(* CoDeSys 2.3.9.42 project: PLC.pro *)
(* Libraries: STANDARD.LIB 5.6.98 12:03:02, TcBase.lib 14.5.09 12:14:08, TcSystem.lib 21.1.15 10:22:54, TcBaseMath.lib 27.7.04 12:07:56, TcMath.lib 23.9.04 15:15:30, TcMC2.lib 6.5.15 08:29:24, TcUtilities.lib 6.1.15 16:45:04, SysLibAlarmTrend.lib 17.10.05 13:12:38 *)

(* Task configuration *)
TASK Standard (PRIORITY := 0, INTERVAL := T#10ms);
	MAIN
END_TASK

(* Global variable list: Global_Variables *)
VAR_GLOBAL
	Flag_FPC_Brd_Err:BOOL;
	Flag_Robot_Alarm:BOOL;

	Total_PauseStatus:BOOL;(*暂停状态*)

	AA: FB_BasicPID;
	MM: BOOL;
	a1: LREAL;
	a2: LREAL;
	OUTPUT:LREAL;

	Process_2_Can_Push2: BOOL;
	Process_2_Can_Push1: BOOL;


	Save_Par:FB_WritePersistentData;
	Save_Button:BOOL;

	Liftin_Feed_1_Run:BOOL;(*喂料1运行触发*)
	Liftin_Feed_Left_1_Run:BOOL;(*喂料1运行触发*)
	Liftin_Feed_Left_2_Run:BOOL;(*喂料1运行触发*)
	Liftin_Feed_Right_1_Run:BOOL;(*喂料1运行触发*)
	Liftin_Feed_Right_2_Run:BOOL;(*喂料1运行触发*)
	Left_Carry_Run:BOOL;(*左搬运*)
	PC_Pause:BOOL;(*上位机给我暂停*)

	Right_Carry_Run:BOOL;(*左搬运*)
	Product_Film_Handel_Run:BOOL;(*吸膜撕膜位置工作触发*)

	Left_Translation_Run:BOOL;(*左平移运行触发*)
	Left_Translation_Run_1: BOOL;
	Left_Translation_Run_2: BOOL;

	Right_Translation_Run:BOOL;(*右平移运动触发*)
	Rolling_Part_Run:BOOL;(*滚压运行触发*)


(*初始化进程*)
	IniRun_Run:BOOL;(*初始化进程触发*)(*-----------------未用-----------------------------*)
	Model_Choose:BOOL;(*模式选择状态*)
	Need_Ini:BOOL;(*需要初始化*)
	IsIniing:BOOL;(*	初始化中*)
	home_backing:BOOL;(*回原点中*)
	runing: BOOL;(*运行中*)

(*上料升降状态信息*)
	Feed_1_Finish:BOOL;(*上料喂料1完成------to上料流程*)

(*撕膜流程为流程1---------------------左移载为流程2--------------------------*)

(*撕膜流程位置状态标志位*)

	Tray1_Have: BOOL; (*1料盘有料*)
	Tray2_Have: BOOL;(*2料盘有料*)

	Process_1_Get_Finish:BOOL;(*喂料1-----拿到料完成----to feed1*)


	Process_1_Push_Finish:BOOL;(*放料完成-----to流程2*)
	Process_1_Push_Finish_Sure:BOOL;(*放料完成-----to流程2*)


	Process_2_Can_Push:BOOL;(*TO---流程1*)

	Positive1_Safe:BOOL;
	Positive2_Safe:BOOL;
	Positive3_Safe:BOOL;
	Positive4_Safe:BOOL;
	Positive_Wait_Safe:BOOL;
(*1------------------------------------------------2*)
(*1------------------------------------------------1*)
(*1------------------------------------------------1*)
(*1------------------------------------------------1*)
(*1------------------------------------------------1*)
(*1------------------------------------------------1*)
(*1------------------------------------------------1*)
(*4------------------------------------------------3*)

	Positive_Camera_Safe1:BOOL;(*拍照位置1安全*)
	Positive_Camera_Safe2:BOOL;(*拍照位置1安全*)
	Positive_Camera_Safe3:BOOL;(*拍照位置1安全*)
	Positive_Camera_Safe4: BOOL;	(* (*拍照位置1安全*) *)

	Positive_Fit_Safe1:BOOL;(*贴合位置1安全*)
	Positive_Fit_Safe2:BOOL;(*贴合位置1安全*)
	Positive_Fit_Safe3:BOOL;(*贴合位置1安全*)
	Positive_Fit_Safe4:BOOL;(*贴合位置1安全*)







	Process_2_Set_Finish1: BOOL;
	Process_2_Set_Finish2: BOOL;

	Wait_Robort2_Touch_Finish:BOOL;(*机械手2贴合完成，关真空吸*)

	Get_Robot1_Get_Finish:BOOL;(*机械手1对取料贴合完成，左移载可动作-------From   机械手1*)
	Robot2_Push_Finish:BOOL;(*机械手2----放料到滚压完成*)

	Feed_2_Finish:BOOL;(*111111111上料喂料2完成 ------TO 机械手1*)
	Get_Robot1_Tray_Empty:BOOL;(*2222222222机械手1取料盘空信号  -------From  机械手1*)
	zuo_ke_jiang:BOOL;(*5555555左可下降*)
	zuo_down_Finish:BOOL;(*1111111判断是否可放*)
	Left_Can_Move: BOOL;(*3333333可以移动*)
	Left_Move_Finish:BOOL;(*4444444移动完成*)

	Feed_3_Finish:BOOL;(*上料喂料3完成------to   机械手3*)
	Get_Robort3_Tray_Full:BOOL;(*机械手3给出，右升降料盘空*)

	Right_Loading_OK:BOOL;(*上空盘ok*)
	Right_Get_Tray_OK:BOOL;(*取空盘完成*)
	Right_Need_Tray:BOOL;(*要空盘信号*)
	Right_Send_Tray_OK:BOOL;(*上空盘完成*)

	you_down_Finish: BOOL;
	you_ke_jiang: BOOL;
	Right_Can_Move:BOOL;
	Right_Move_Finish:BOOL;



(*滚压流程3---------------------------------------右移载流程4*)

	Process_3_Can_Push:BOOL;(*滚压可放料------to 机械收2*)
	Wait_Robot_Push:BOOL;(*机械手放滚压，开真空吸*)
  	Process_3_Set_Finish:BOOL;(*滚压送出料----完成信号*)

	Process_4_Can_Push:BOOL;(*右移载可放料-------to 滚压流程*)
	Process_4_Set_Finish:BOOL;(*右移载，到位，机械手3可操作------to 机械手3*)
	Get_Robort_simo_Finish: BOOL;(*获取机械手撕膜完成信号*)
	Set_Robort_Can_Get: BOOL;(*告知机械手可取料*)


	Get_Robot3_Get_Finish:BOOL;(*机械手3----给出，取右移载完成信号*)



(*界面按钮*)
	Silencer_Button: BOOL;(*消音按钮*)
	Discharge_Button:BOOL;(*排料按钮*)

	UP_Button:BOOL;(*上料按钮*)
	Left_UP_Button:BOOL;(*左上料按钮*)
	Left_Down_Button:BOOL;(*右卸料按钮*)

	Right_UP_Button:BOOL;(*右上料按钮*)
	Right_Down_Button:BOOL;(*右卸料按钮*)

	Button_Ad:BOOL;

	Feed1_Button:BOOL;(*上料自动按钮*)
	Feed_Left_Button1:BOOL;(*左上升自动按钮*)
	Feed_Left_Button2:BOOL;(*左下降自动按钮*)
	Feed_Right_Button1:BOOL;(*右上升自动按钮*)
	Feed_Right_Button2:BOOL;(*右下降自动按钮*)





(*显示运行状态*)




(*显示报警*)


(*标志位1*)
	shou_have_mo:BOOL;(*有膜*)
	shou_have_moliao:BOOL;(*有膜料*)
	shou_have_liao:BOOL;(*有料*)
	zai_have_liao:BOOL;(*载盘有料*)
	zai_have_mo:BOOL;(*载盘有膜*)


(*接收机械手完成信号*)
	Camera_1_1_OK:BOOL;(*已拍照1-----FROM JIXIESHOU*)
	Camera_1_2_OK:BOOL;(*已拍照2-----FROM JIXIESHOU*)
	Camera_1_3_OK:BOOL;(*已拍照3-----FROM JIXIESHOU*)
	Camera_1_4_OK:BOOL;(*已拍照4-----FROM JIXIESHOU*)

	Camera_2_1_OK:BOOL;(*已拍照1-----FROM JIXIESHOU*)
	Camera_2_2_OK:BOOL;(*已拍照2-----FROM JIXIESHOU*)



(*左流程，运行触发----发送给机械手*)
	Camera_1_1_run:BOOL;(*拍照1标志位-----TO JIXIESOU*)
	Camera_1_2_run:BOOL;(*拍照2标志位----TO JIXIESOU*)
	Camera_1_3_run:BOOL;(*拍照3标志位----TO JIXIESOU*)
	Camera_1_4_run:BOOL;(*拍照4标志位----TO JIXIESOU*)
	Camera_2_1_run:BOOL;(*拍照1标志位-----TO JIXIESOU*)
	Camera_2_2_run:BOOL;(*拍照2标志位----TO JIXIESOU*)

	Camera_1_5_run: BOOL;
	Camera_1_5_OK: BOOL;
	Camera_1_6_run: BOOL;
	Camera_1_6_OK: BOOL;
	Camera_1_7_run: BOOL;
	Camera_1_7_OK: BOOL;
	Camera_1_8_run: BOOL;
	Camera_1_8_OK: BOOL;

	FG_Ready_1:BOOL;
	FG_Ready_2:BOOL;
	FG_Ready_3:BOOL;
	FG_Ready_4:BOOL;
	FG_Ready_5:BOOL;
	FG_Ready_6:BOOL;
	FG_Ready_7:BOOL;
	FG_Ready_8:BOOL;

	HB_Fit_Finish_1:BOOL;
	HB_Fit_Finish_2:BOOL;
	HB_Fit_Finish_3:BOOL;
	HB_Fit_Finish_4:BOOL;
	HB_Fit_Finish_5:BOOL;
	HB_Fit_Finish_6:BOOL;
	HB_Fit_Finish_7: BOOL;
	HB_Fit_Finish_8: BOOL;

	Can_Move_Film:BOOL;



(*左流程，各状态位*)

	paizhao1_OK:BOOL;
	paizhao2_OK:BOOL;
	paizhao3_OK:BOOL;
	paizhao4_OK:BOOL;
	pan_have_liao2:BOOL;(*载盘右有料*)
	paizhao2_1_OK:BOOL;
	paizhao2_2_OK:BOOL;

(*滚压流程标志位*)
	rolling_have_liao:BOOL;(*滚压盘有料状态*)
	Rolling_Number:INT;(*关压次数*)


(*左搬运状态标志位*)
	Left_hand_have:BOOL;(*左收手上有料*)
	Right_hand_have:BOOL;(*右收手上有料*)


	No_need_Pause1: BOOL;
	No_need_Pause2: BOOL;

	Empty_Pro:BOOL;(*空跑程序，触发信号*)
	All_Rset: BOOL;
	All_Start:BOOL;
	All_Stop:BOOL;






END_VAR

(* Global variable list: Global_Variables_Alam *)
VAR_GLOBAL

	Total_Axis_Error: BOOL;
	Axis1_Error:BOOL;
	Axis2_Error:BOOL;
	Axis3_Error:BOOL;
	Axis4_Error:BOOL;
	Axis5_Error:BOOL;
	Axis6_Error:BOOL;
	Axis7_Error:BOOL;
	Axis8_Error:BOOL;
	Axis9_Error:BOOL;
	Axis10_Error:BOOL;
	Axis11_Error:BOOL;











	Total_Emergency:BOOL;(*总急停*)
	Axis1_Limit_Emergency:BOOL;(*轴1限位急停*)
	Axis2_Limit_Emergency:BOOL;
	Axis3_Limit_Emergency:BOOL;
	Axis4_Limit_Emergency:BOOL;
	Axis5_Limit_Emergency:BOOL;
	Axis6_Limit_Emergency:BOOL;
	Axis7_Limit_Emergency:BOOL;
	Axis8_Limit_Emergency:BOOL;
	Axis9_Limit_Emergency: BOOL;	(*  *)
	Axis10_Limit_Emergency: BOOL;	(*  *)
	Axis11_Limit_Emergency: BOOL;	(*  *)

	Motion_Alam_Rst:BOOL;(*伺服报警复位*)

	Total_Pause:BOOL;(*总暂停*)

	Pressure_Fail_1:BOOL;(*撕膜负压失败*)
	Pressure_Fail_2:BOOL;(*撕膜取料负压失败*)

	UP_Down_Alam1: BOOL;
	UP_Down_Alam2: BOOL;


	Left_Cylinder_Alam_1:BOOL;(*左升降，平移气缸报警*)
	Left_Cylinder_Alam_2:BOOL;(*左升降，上下气缸报警*)
	Pressure_Left_Fail:BOOL;(*左升降，负压吸取失败*)

	Right_Cylinder_Alam_1:BOOL;(*右升降，平移气缸报警*)
	Right_Cylinder_Alam_2:BOOL;(*右升降，上下气缸报警*)
	Pressure_Right_Fail:BOOL;(*右升降，负压吸取失败*)

	Rolling_Cylinder_Alam_1:BOOL;(*滚压推入气缸报警*)
	Rolling_Cylinder_Alam_2:BOOL;(*滚压上下气缸报警*)
	Rolling_Cylinder_Alam_3:BOOL;(*滚压翻转气缸报警*)
	Rolling_Pressure_Fail:BOOL;(*滚压负压表报警*)

	Feed_1_Nome_Alam:BOOL;(*上料空报警*)
	Feed_Left_None_Alam:BOOL;(*左上无料*)
	Feed_Left_Full_Alam:BOOL;(*左下料满*)
	Feed_Right_None_Alam:BOOL;(*右上无料*)
	Feed_Right_Full_Alam:BOOL;(*右上料满*)



	Total_Door_Alam:BOOL;(*门报警*)
	Door1_Alam:BOOL;(*门1报警*)
	Door2_Alam:BOOL;(*门1报警*)
	Door3_Alam:BOOL;(*门1报警*)
	Door4_Alam:BOOL;(*门1报警*)

	Power_Door1: BOOL;
	Power_Door2: BOOL;
	Power_Door3: BOOL;
	Passtray_Door: BOOL;
	HB_Door1: BOOL;
	HB_Door2: BOOL;

	No_need_Pause:BOOL;

	Shield_Door:BOOL:=TRUE;(*屏蔽安全门*)

	No_Feed_1:BOOL;(*撕膜位置上料物料提示*)

	No_Feed_Left_Up:BOOL;(*左上升位置上料物料提示*)
	No_Feed_Left_Down:BOOL;(*左下降位置上料物料提示*)

	No_Feed_Right_Up:BOOL;(*右上升位置上料物料提示*)
	No_Feed_Right_Down:BOOL;(*右下降下降位置上料物料提示*)

	Message: ARRAY [0..messagenum] 		OF BOOL;  (*运行信息数组*)
	PC_Message:ARRAY[0..pc_messagenum] OF BOOL;(*pc显示使用*)
	Alam: ARRAY [0..alamnum] 		OF BOOL; (*报警信息数组*)

	Camera1_NG:BOOL;(*F&G拍照NG*)
	Camera2_NG:BOOL;(*FPC拍照NG*)
	Camera1_NG_Pause: BOOL;(*暂停状态*)

	Feed1_UnReady: BOOL;(*FG上料为到位*)
	FPC_up_Unready: BOOL;
	FPC_down_Unready: BOOL;
	TRAY_up_Unready: BOOL;
	TRAY_down_Unready: BOOL;

END_VAR

VAR_GLOBAL CONSTANT
	messagenum:UINT := 300;
	alamnum:UINT := 300;
	pc_messagenum:UINT:=300;


END_VAR

(* Global variable list: Global_Variables_Axis *)
VAR_GLOBAL
(*轴定义*)
 	Axis1:AXIS_REF;   (*左移载*)
	Axis2:AXIS_REF;   (*右移载*)
	Axis3:AXIS_REF;   (*上料升降电机*)
	Axis4:AXIS_REF;   (*上料移载电机*)
	Axis5:AXIS_REF;   (*上料撕膜取料电机*)
	Axis6:AXIS_REF;   (*左上升电机*)
	Axis7:AXIS_REF;   (*左下降电机*)
	Axis8:AXIS_REF;   (*右上升电机*)
	Axis9:AXIS_REF;   (*右下降电机*)
	Axis10:AXIS_REF;   (*滚压电机*)
	Axis11:AXIS_REF;(*左移载2*)


(*轴使能*)
	Axis1_Poweron:BOOL;(*左移电机使能*)
	Axis2_Poweron: BOOL;	(*右移电机使能*)
	Axis3_Poweron: BOOL;	 (*上料升降电机使能*)
	Axis4_Poweron:BOOL;(*上料移载电机使能*)
	Axis5_Poweron:BOOL;(*上料撕膜取料电机使能*)
	Axis6_Poweron:BOOL;(*左上升电机使能*)
	Axis7_Poweron:BOOL;(*左下降电机使能*)
	Axis8_Poweron:BOOL;(*右上升电机使能*)
	Axis9_Poweron: BOOL;	(*右下降电机使能*)
	Axis10_Poweron:BOOL;(*滚压电机使能*)
	Axis11_Poweron:BOOL;(*左移载2使能*)


(*回原点*)
	Axis1_Home:BOOL;(*左移电机回原*)
	Axis2_Home: BOOL;	(*右移电机回原*)
	Axis3_Home: BOOL;	 (*上料升降电机回原*)
	Axis4_Home:BOOL;(*上料移载电机回原*)
	Axis5_Home:BOOL;(*上料撕膜取料电机回原*)
	Axis6_Home:BOOL;(*左上升电机回原*)
	Axis7_Home:BOOL;(*左下降电机回原*)
	Axis8_Home:BOOL;(*右上升电机回原*)
	Axis9_Home: BOOL;	(*右下降电机回原*)
	Axis10_Home:BOOL;(*滚压电机回原*)
	Axis11_Home:BOOL;(*左移载电机回原2*)

(*PTF*)

	Axis1_PTF:BOOL;(*左移电机持续运动*)
	Axis2_PTF: BOOL;	(*右移电机持续运动*)
	Axis3_PTF: BOOL;	 (*上料升降电机持续运动*)
	Axis4_PTF:BOOL;(*上料移载电机持续运动*)
	Axis5_PTF:BOOL;(*上料撕膜取料电机持续运动*)
	Axis6_PTF:BOOL;(*左上升电机持续运动*)
	Axis7_PTF:BOOL;(*左下降电机持续运动*)
	Axis8_PTF:BOOL;(*右上升电机持续运动*)
	Axis9_PTF: BOOL;	(*右下降电机迟训运动*)
	Axis10_PTF:BOOL;(*滚压电机持续运动*)
	Axis11_PTF:BOOL;(*左移载电机持续运动2*)



	Axis3_PTF_2: BOOL;
	Axis6_PTF_2: BOOL;
	Axis7_PTF_2: BOOL;
	Axis8_PTF_2: BOOL;
	Axis9_PTF_2: BOOL;

(*Halt*)

	Axis1_Halt:BOOL;(*左移电机停止*)
	Axis2_Halt: BOOL;	(*右移电机停止*)
	Axis3_Halt: BOOL;	 (*上料升降电机停止*)
	Axis4_Halt:BOOL;(*上料移载电机停止*)
	Axis5_Halt:BOOL;(*上料撕膜取料电机停止*)
	Axis6_Halt:BOOL;(*左上升电机持停止*)
	Axis7_Halt:BOOL;(*左下降电机停止*)
	Axis8_Halt:BOOL;(*右上升电机持停止*)
	Axis9_Halt: BOOL;	(*右下降电机停止*)
	Axis10_Halt:BOOL;(*滚压电机停止*)
	Axis11_Halt:BOOL;(*左移载电机停止2*)

(*绝对位置*)

	Axis1_MoveAbsolute:BOOL;(*左移电机绝对位置*)
	Axis2_MoveAbsolute: BOOL;	(*右移电机绝对位置*)
	Axis3_MoveAbsolute: BOOL;	 (*上料升降电机绝对位置*)
	Axis4_MoveAbsolute:BOOL;(*上料移载电机绝对位置*)
	Axis5_MoveAbsolute:BOOL;(*上料撕膜取料电机绝对位置*)
	Axis6_MoveAbsolute:BOOL;(*左上升电机持绝对位置*)
	Axis7_MoveAbsolute:BOOL;(*左下降电机绝对位置*)
	Axis8_MoveAbsolute:BOOL;(*右上升电机持绝对位置*)
	Axis9_MoveAbsolute: BOOL;	(*右下降电机绝对位置*)
	Axis10_MoveAbsolute:BOOL;(*滚压电机绝对位置*)
	Axis11_MoveAbsolute:BOOL;(*左移载电机绝对位置2*)


	Axis4_1_MoveAbsolute: BOOL;
	Axis5_1_MoveAbsolute: BOOL;
	Axis10_MoveAbsolute1: BOOL;






END_VAR

(* Global variable list: Global_Variables_Axis_13X *)
VAR_GLOBAL
	Axis13:AXIS_REF;(*左移载2*)
	Axis13_Poweron:BOOL;(*左移载2使能*)
	Axis13_Home:BOOL;(*左移电机回原*)
	Axis13_PTF:BOOL;(*左移电机持续运动*)
	Axis13_Halt:BOOL;(*左移电机停止*)
	Axis13_MoveAbsolute:BOOL;(*左移电机绝对位置*)


	Axis13_Error:BOOL;
	Axis13_Limit_Emergency:BOOL;(*轴1限位急停*)

	Axis13_Home_Function: MC_Home;
	Axis13_Power_Function: MC_Power;
	Axis13_Abs_Function: MC_MoveAbsolute;
	Axis13_PTF_Function: MC_MoveVelocity;
	Axis13_Halt_Function: MC_Halt;
	Axis13_Rst_Function: MC_Reset;


	Axis13_debug_trigger:BOOL;(*电机1调试模式触发*)
	Axis13_mov_add:BOOL;(*轴1加*)
	Axis13_mov_sub:BOOL;(*轴1减*)
	Axis13_mov_line:BOOL;(*轴1运动到点*)
	D213:LREAL;(*调试轴12运动到点*)

	Axis13_Positive_Limit: BOOL;
	Axis13_Negative_Limit: BOOL;
	Axis13_BackHome_trigger:BOOL;
	Axis13_Negative_Invalid:BOOL;
	Axis13_BackHome_OK:BOOL;


	D1_3:LREAL;(*轴12位置*)
	D2_3:LREAL;(*轴12速度*)



END_VAR

VAR_GLOBAL PERSISTENT
	A13_W0:LREAL;(*初始位置----回的位置*)
	A13_W1:LREAL;(*压合上位置*)
	A13_W2:LREAL;(*压合下位置*)


END_VAR

(* Global variable list: Global_Variables_Axis_Rolling *)
VAR_GLOBAL
	Axis12:AXIS_REF;(*左移载2*)

	Axis12_Poweron:BOOL;(*左移载2使能*)
	Axis12_Home:BOOL;(*左移电机回原*)
	Axis12_PTF:BOOL;(*左移电机持续运动*)
	Axis12_Halt:BOOL;(*左移电机停止*)
	Axis12_MoveAbsolute:BOOL;(*左移电机绝对位置*)


	Axis12_Error:BOOL;
	Axis12_Limit_Emergency:BOOL;(*轴1限位急停*)

	Axis12_Home_Function: MC_Home;
	Axis12_Power_Function: MC_Power;
	Axis12_Abs_Function: MC_MoveAbsolute;
	Axis12_PTF_Function: MC_MoveVelocity;
	Axis12_Halt_Function: MC_Halt;
	Axis12_Rst_Function: MC_Reset;


	Axis12_debug_trigger:BOOL;(*电机1调试模式触发*)
	Axis12_mov_add:BOOL;(*轴1加*)
	Axis12_mov_sub:BOOL;(*轴1减*)
	Axis12_mov_line:BOOL;(*轴1运动到点*)
	D212:LREAL;(*调试轴12运动到点*)

	Axis12_Positive_Limit: BOOL;
	Axis12_Negative_Limit: BOOL;
	Axis12_BackHome_trigger:BOOL;
	Axis12_Negative_Invalid:BOOL;
	Axis12_BackHome_OK:BOOL;


	D1_2:LREAL;(*轴12位置*)
	D2_2:LREAL;(*轴12速度*)
	F_push AT %I*: INT;(*压力传感器传入数据*)


END_VAR

VAR_GLOBAL PERSISTENT
	A12_W0:LREAL;(*初始位置----回的位置*)
	A12_W1:LREAL;(*压合上位置*)
	A12_W2:LREAL;(*压合下位置*)


END_VAR

(* Global variable list: Global_Variables_AxisFun *)
VAR_GLOBAL
(*回原点功能块*)
	Axis1_Home_Function: MC_Home;
	Axis2_Home_Function: MC_Home;
	Axis3_Home_Function: MC_Home;
	Axis4_Home_Function: MC_Home;
	Axis5_Home_Function: MC_Home;
	Axis6_Home_Function: MC_Home;
	Axis7_Home_Function: MC_Home;
	Axis8_Home_Function: MC_Home;
	Axis9_Home_Function: MC_Home;
	Axis10_Home_Function: MC_Home;
	Axis11_Home_Function: MC_Home;


(*使能功能块*)
	Axis1_Power_Function: MC_Power;
	Axis2_Power_Function: MC_Power;
	Axis3_Power_Function: MC_Power;
	Axis4_Power_Function: MC_Power;
	Axis5_Power_Function: MC_Power;
	Axis6_Power_Function: MC_Power;
	Axis7_Power_Function: MC_Power;
	Axis8_Power_Function: MC_Power;
	Axis9_Power_Function: MC_Power;
	Axis10_Power_Function: MC_Power;
	Axis11_Power_Function: MC_Power;

(*绝对位置功能块*)
	Axis1_Abs_Function: MC_MoveAbsolute;
	Axis2_Abs_Function: MC_MoveAbsolute;
	Axis3_Abs_Function: MC_MoveAbsolute;
	Axis4_Abs_Function: MC_MoveAbsolute;
	Axis5_Abs_Function: MC_MoveAbsolute;
	Axis6_Abs_Function: MC_MoveAbsolute;
	Axis7_Abs_Function: MC_MoveAbsolute;
	Axis8_Abs_Function: MC_MoveAbsolute;
	Axis9_Abs_Function: MC_MoveAbsolute;
	Axis10_Abs_Function: MC_MoveAbsolute;
	Axis11_Abs_Function: MC_MoveAbsolute;


	Axis10_Abs_Function1: MC_MoveAbsolute;
	Axis5_1_Abs_Function: MC_MoveAbsolute;
	Axis4_1_Abs_Function: MC_MoveAbsolute;



(*PTF*)
	Axis1_PTF_Function: MC_MoveVelocity;
	Axis2_PTF_Function: MC_MoveVelocity;
	Axis3_PTF_Function: MC_MoveVelocity;
	Axis4_PTF_Function: MC_MoveVelocity;
	Axis5_PTF_Function: MC_MoveVelocity;
	Axis6_PTF_Function: MC_MoveVelocity;
	Axis7_PTF_Function: MC_MoveVelocity;
	Axis8_PTF_Function: MC_MoveVelocity;
	Axis9_PTF_Function: MC_MoveVelocity;
	Axis10_PTF_Function: MC_MoveVelocity;
	Axis11_PTF_Function: MC_MoveVelocity;

	Axis3_PTF_Function_2: MC_MoveVelocity;
	Axis6_PTF_Function_2: MC_MoveVelocity;
	Axis7_PTF_Function_2: MC_MoveVelocity;
	Axis8_PTF_Function_2: MC_MoveVelocity;
	Axis9_PTF_Function_2: MC_MoveVelocity;

(*Halt*)
	Axis1_Halt_Function: MC_Halt;
	Axis2_Halt_Function: MC_Halt;
	Axis3_Halt_Function: MC_Halt;
	Axis4_Halt_Function: MC_Halt;
	Axis5_Halt_Function: MC_Halt;
	Axis6_Halt_Function: MC_Halt;
	Axis7_Halt_Function: MC_Halt;
	Axis8_Halt_Function: MC_Halt;
	Axis9_Halt_Function: MC_Halt;
	Axis10_Halt_Function: MC_Halt;
	Axis11_Halt_Function: MC_Halt;


(*RSET*)

	Axis1_Rst_Function: MC_Reset;
	Axis2_Rst_Function: MC_Reset;
	Axis3_Rst_Function: MC_Reset;
	Axis4_Rst_Function: MC_Reset;
	Axis5_Rst_Function: MC_Reset;
	Axis6_Rst_Function: MC_Reset;
	Axis7_Rst_Function: MC_Reset;
	Axis8_Rst_Function: MC_Reset;
	Axis9_Rst_Function: MC_Reset;
	Axis10_Rst_Function: MC_Reset;
	Axis11_Rst_Function: MC_Reset;

END_VAR

(* Global variable list: Global_Variables_Coord *)
VAR_GLOBAL

	D1:LREAL;(*轴1位置*)
	D11:LREAL;(*轴1速度*)

	D2:LREAL;(*轴2位置*)
	D12:LREAL;(*轴2速度*)

	D3:LREAL;(*轴3位置*)
	D13:LREAL;(*轴3速度*)

	D4:LREAL;(*轴4位置*)
	D14:LREAL;(*轴4速度*)

	D5:LREAL;(*轴5位置*)
	D15:LREAL;(*轴5速度*)

	D6:LREAL;(*轴6位置*)
	D16:LREAL;(*轴6速度*)

	D7:LREAL;(*轴7位置*)
	D17:LREAL;(*轴7速度*)

	D8:LREAL;(*轴8位置*)
	D18:LREAL;(*轴8速度*)

	D9:LREAL;(*轴9位置*)
	D19:LREAL;(*轴9速度*)

	D10:LREAL;(*轴10位置*)
	D20:LREAL;(*轴10速度*)

	D1_1:LREAL;(*轴11位置*)
	D2_1:LREAL;(*轴11速度*)

	D14_1: LREAL;
	D15_1: LREAL;


	D10_1: LREAL;





	M100:BOOL;(*低速设置信号*)
	M101:BOOL;(*中速设置信号*)
	M102:BOOL;(*高速设置信号*)

END_VAR



VAR_GLOBAL PERSISTENT
(*调速寄存及信号*)

	D100: ARRAY [0..11] 		OF LREAL;   (*低速*)
	D101: ARRAY [0..11] 		OF LREAL;   (*中速*)
	D102: ARRAY [0..11] 		OF LREAL;   (*高速*)

	D103: ARRAY [0..11] 		OF LREAL;   (*当前位置监控*)

END_VAR

VAR_GLOBAL PERSISTENT
(*运行坐标*)
	D300:LREAL;(*Axis3----进料喂料电机初始位置*)(*下面位置-----当空料盘后，回到初始位置*)

	D600:LREAL;(*Axis6-----左上升料喂料电机初始位置*)(*下面位置-----当空料盘后，回到初始位置*)

	D700:LREAL;(*Axis7-----左下降喂料电机初始位置*)(*下面位置-----当空料盘后，回到初始位置*)
	D710:LREAL;(*Axis7-----左下降喂料电机初始位置*)(*下面位置-----当空料盘后，回到初始位置*)

	D800:LREAL;(*Axis8-----右上升喂料电机初始位置*)(*上面位置-----当空料盘后，回到初始位置*)
	D810:LREAL;(*Axis9-----右下降喂料电机初始位置*)(*下面位置-----当空料盘后，回到初始位置*)

	D900:LREAL;(*Axis9-----右下降喂料电机初始位置*)(*下面位置-----当空料盘后，回到初始位置*)
	D910:LREAL;(*Axis9-----右下降喂料电机初始位置*)(*下面位置-----当空料盘后，回到初始位置*)


	(*Axis4-------水平移动移载电机*)
	A4_W0:LREAL;(*初始位置*)
	A4_W1:LREAL;(*取料工位-----初始位置*)
	A4_W2:LREAL;(*撕膜平台工位*)
	A4_W3:LREAL;(*丢膜工位*)
	A4_W4:LREAL;(*放料工位*)
	A4_W5:LREAL;(*撕膜联动X位置*)

	(*Axis5-------撕膜电机-加吸料*)
	A5_W0:LREAL;(*初始位置*)
	A5_W1:LREAL;(*取料下降工位*)
	A5_W2:LREAL;(*撕膜平台下降工位*)
	A5_W3:LREAL;(*丢膜下降工位*)
	A5_W4:LREAL;(*放料下降工位*)
	A5_W5:LREAL;(*撕膜Z轴上抬一点*)
	A5_W6:LREAL;(*撕膜联动位置Z*)
	A5_W7:LREAL;(*完成送料上抬一点位置*)
	A5_W8: LREAL;(*联动之后上抬节点*)






	(*Axis10-------滚压电机-*)
	A10_W0:LREAL;(*初始位置----回的位置*)
	A10_W1:LREAL;(*滚压进到位工位*)
	A10_W2:LREAL;(*滚压回到位工位*)

	(*Axis1-------左移载电机-*)
	A1_W0:LREAL;(*初始位置----回的位置*)
	A1_W1:LREAL;(*等待放料位置*)

	A1_W2:LREAL;(*拍照1*)
	A1_W3:LREAL;(*拍照2*)
	A1_W4:LREAL;(*拍照3*)
	A1_W5:LREAL;(*拍照4*)

	A1_W6:LREAL;(*贴合工位1*)
	A1_W7:LREAL;(*贴合工位2*)
	A1_W8:LREAL;(*贴合工位3*)
	A1_W9:LREAL;(*贴合工位4*)

	A1_W10:LREAL;(*循环位置2位置*)
	DTest0: ARRAY [0..10] 		OF LREAL;   (*当前位置监控*)
	DTest10: ARRAY [0..10] 		OF LREAL;   (*当前位置监控*)

	Debug1:ARRAY[0..3] OF LREAL;







	A11_W0:LREAL;(*初始位置----回的位置*)
	A11_W1:LREAL;(*等待放料位置*)
	A11_W2:LREAL;(*拍照1*)
	A11_W3:LREAL;(*拍照2*)
	A11_W4:LREAL;(*拍照3*)
	A11_W5:LREAL;(*拍照4*)

	A11_W6:LREAL;(*贴合工位1*)
	A11_W7:LREAL;(*贴合工位2*)
	A11_W8:LREAL;(*贴合工位3*)
	A11_W9:LREAL;(*贴合工位4*)



	A11_W10:LREAL;(*循环位置2位置*)

	DTest: ARRAY [0..10] 		OF LREAL;   (*当前位置监控*)
	DTest00: ARRAY [0..10] 		OF LREAL;   (*当前位置监控*)

	Debug2:ARRAY[0..3] OF LREAL;


	(*Axis2-------左移载电机-*)
	A2_W0:LREAL;(*初始位置----回的位置*)
	A2_W1:LREAL;(*滚压等待扣料位置*)
	A2_W2:LREAL;(*扫码位置1*)
	A2_W3:LREAL;(*扫码位置2*)
	A2_W4:LREAL;(*排淬等待位置*)

	Set_Rolling_Number:LREAL;(*设置的压合次数*)

	D20_1: LREAL;(*滚压速度设置*)

	RollTime: LREAL;(*滚压时间显示*)
END_VAR

(* Global variable list: Global_Variables_Debug *)
VAR_GLOBAL
	Debug_Model:BOOL; (*调试模信号*)
	debug_FLIG: BOOL;

	Axis1_debug_trigger:BOOL;(*电机1调试模式触发*)
	Axis2_debug_trigger:BOOL;(*电机1调试模式触发*)
	Axis3_debug_trigger:BOOL;(*电机1调试模式触发*)
	Axis4_debug_trigger:BOOL;(*电机1调试模式触发*)
	Axis5_debug_trigger:BOOL;(*电机1调试模式触发*)
	Axis6_debug_trigger:BOOL;(*电机1调试模式触发*)
	Axis7_debug_trigger:BOOL;(*电机1调试模式触发*)
	Axis8_debug_trigger:BOOL;(*电机1调试模式触发*)
	Axis9_debug_trigger:BOOL;(*电机1调试模式触发*)
	Axis10_debug_trigger:BOOL;(*电机10调试模式触发*)
	Axis11_debug_trigger:BOOL;(*电机11调试模式触发*)
	Others_debug_trigger:BOOL;(*电机1调试模式触发*)

	D200:LREAL;(*点动距离*)

	Axis1_mov_add:BOOL;(*轴1加*)
	Axis1_mov_sub:BOOL;(*轴1减*)
	Axis1_mov_line:BOOL;(*轴1运动到点*)
	D201:LREAL;(*调试轴1运动到点*)

	Axis2_mov_add:BOOL;(*轴1加*)
	Axis2_mov_sub:BOOL;(*轴1减*)
	Axis2_mov_line:BOOL;(*轴1运动到点*)
	D202:LREAL;(*调试轴1运动到点*)

	Axis3_mov_add:BOOL;(*轴1加*)
	Axis3_mov_sub:BOOL;(*轴1减*)
	Axis3_mov_line: BOOL;	(* (*轴1运动到点*) *)
	D203:LREAL;(*调试轴1运动到点*)

	Axis4_mov_add:BOOL;(*轴1加*)
	Axis4_mov_sub:BOOL;(*轴1减*)
	Axis4_mov_line:BOOL;(*轴1运动到点*)
	D204:LREAL;(*调试轴1运动到点*)

	Axis5_mov_add:BOOL;(*轴1加*)
	Axis5_mov_sub:BOOL;(*轴1减*)
	Axis5_mov_line:BOOL;(*轴1运动到点*)
	D205:LREAL;(*调试轴1运动到点*)

	Axis6_mov_add:BOOL;(*轴1加*)
	Axis6_mov_sub:BOOL;(*轴1减*)
	Axis6_mov_line:BOOL;(*轴1运动到点*)
	D206:LREAL;(*调试轴1运动到点*)

	Axis7_mov_add:BOOL;(*轴1加*)
	Axis7_mov_sub:BOOL;(*轴1减*)
	Axis7_mov_line:BOOL;(*轴1运动到点*)
	D207:LREAL;(*调试轴1运动到点*)

	Axis8_mov_add:BOOL;(*轴1加*)
	Axis8_mov_sub:BOOL;(*轴1减*)
	Axis8_mov_line:BOOL;(*轴1运动到点*)
	D208:LREAL;(*调试轴1运动到点*)

	Axis9_mov_add:BOOL;(*轴1加*)
	Axis9_mov_sub:BOOL;(*轴1减*)
	Axis9_mov_line:BOOL;(*轴1运动到点*)
	D209:LREAL;(*调试轴1运动到点*)

	Axis10_mov_add:BOOL;(*轴1加*)
	Axis10_mov_sub:BOOL;(*轴1减*)
	Axis10_mov_line:BOOL;(*轴1运动到点*)
	D210:LREAL;(*调试轴1运动到点*)

	Axis11_mov_add:BOOL;(*轴1加*)
	Axis11_mov_sub:BOOL;(*轴1减*)
	Axis11_mov_line:BOOL;(*轴1运动到点*)
	D211:LREAL;(*调试轴1运动到点*)







END_VAR

(* Global variable list: Global_Variables_Home_Back *)
VAR_GLOBAL

	Axis1_Positive_Limit: BOOL;
	Axis1_Negative_Limit: BOOL;
	Axis2_Positive_Limit: BOOL;
	Axis2_Negative_Limit: BOOL;
	Axis3_Negative_Limit: BOOL;
	Axis3_Positive_Limit: BOOL;
	Axis4_Positive_Limit: BOOL;
	Axis4_Negative_Limit: BOOL;
	Axis5_Positive_Limit: BOOL;
	Axis5_Negative_Limit: BOOL;
	Axis6_Positive_Limit: BOOL;
	Axis6_Negative_Limit: BOOL;
	Axis7_Positive_Limit: BOOL;
	Axis7_Negative_Limit: BOOL;
	Axis8_Positive_Limit: BOOL;
	Axis8_Negative_Limit: BOOL;
	Axis9_Positive_Limit: BOOL;
	Axis9_Negative_Limit: BOOL;
	Axis10_Positive_Limit: BOOL;
	Axis10_Negative_Limit: BOOL;
	Axis11_Positive_Limit: BOOL;
	Axis11_Negative_Limit: BOOL;

(*轴回原触发*)
	Axis1_BackHome_trigger:BOOL;
	Axis2_BackHome_trigger:BOOL;
	Axis3_BackHome_trigger:BOOL;
	Axis4_BackHome_trigger:BOOL;
	Axis5_BackHome_trigger:BOOL;
	Axis6_BackHome_trigger: BOOL;	(*  *)
	Axis7_BackHome_trigger:BOOL;
	Axis8_BackHome_trigger:BOOL;
	Axis9_BackHome_trigger: BOOL;	(*  *)
	Axis10_BackHome_trigger: BOOL;	(*  *)
	Axis11_BackHome_trigger: BOOL;	(*  *)

(*轴反极限无效*)
	Axis1_Negative_Invalid:BOOL;
	Axis2_Negative_Invalid:BOOL;
	Axis3_Negative_Invalid:BOOL;
	Axis4_Negative_Invalid:BOOL;
	Axis5_Negative_Invalid:BOOL;
	Axis6_Negative_Invalid:BOOL;
	Axis7_Negative_Invalid:BOOL;
	Axis8_Negative_Invalid:BOOL;
	Axis9_Negative_Invalid:BOOL;
	Axis10_Negative_Invalid:BOOL;
	Axis11_Negative_Invalid:BOOL;


(*轴回原OK*)
	Axis1_BackHome_OK:BOOL;
	Axis2_BackHome_OK:BOOL;
	Axis3_BackHome_OK:BOOL;
	Axis4_BackHome_OK:BOOL;
	Axis5_BackHome_OK:BOOL;
	Axis6_BackHome_OK:BOOL;
	Axis7_BackHome_OK:BOOL;
	Axis8_BackHome_OK:BOOL;
	Axis9_BackHome_OK:BOOL;
	Axis10_BackHome_OK:BOOL;
	Axis11_BackHome_OK:BOOL;

END_VAR

(* Global variable list: Global_Variables_io *)
VAR_GLOBAL


(*EL1889-0*)
	X0_1 AT %I*: BOOL; (*送料上升正极限*)
	X0_2 AT %I*: BOOL; (*送料上升原点*)
	X0_3 AT %I*: BOOL; (*送料上升反极限*)
	X0_4 AT %I*: BOOL; (*送料移载正极限*)
	X0_5 AT %I*: BOOL; (*送料移载原点*)
	X0_6 AT %I*: BOOL; (*送料移载反极限*)
	X0_7 AT %I*: BOOL; (*送料撕膜正极限*)
	X0_8 AT %I*: BOOL; (*送料撕膜原点*)
	X0_9 AT %I*: BOOL; (*送料撕膜反极限*)
	X0_10 AT %I*: BOOL; (*左送料上升正极限*)
	X0_11 AT %I*: BOOL; (*左送料上升原点*)
	X0_12 AT %I*: BOOL; (*左送料上升反极限*)
	X0_13 AT %I*: BOOL; (*左收盘下降正极限*)
	X0_14 AT %I*: BOOL; (*左送盘下降原点*)
	X0_15 AT %I*: BOOL; (*左送盘下降反极限*)
	X0_16 AT %I*: BOOL; (*左移载正极限*)


(*EL1889-1*)
	X1_1 AT %I*: BOOL; (*左移载原点*)
	X1_2 AT %I*: BOOL; (*左移载反极限*)
	X1_3 AT %I*: BOOL; (*右送盘上升正极限*)
	X1_4 AT %I*: BOOL; (*右送盘上升原点*)
	X1_5 AT %I*: BOOL; (*右送盘上升反极限*)
	X1_6 AT %I*: BOOL; (*右收料下降正极限*)
	X1_7 AT %I*: BOOL; (*右收料下降原点*)
	X1_8 AT %I*: BOOL; (*右收料下降反极限*)
	X1_9 AT %I*: BOOL; (*右移载正极限*)
	X1_10 AT %I*: BOOL;  (*右移载原点*)
	X1_11 AT %I*: BOOL; (*右移载反极限*)
	X1_12 AT %I*: BOOL; (*滚压正极限*)
	X1_13 AT %I*: BOOL; (*滚压原点*)
	X1_14 AT %I*: BOOL; (*滚压反极限*)
	X1_15 AT %I*: BOOL;(*FPC上升到位传感器-----------*)
	X1_16 AT %I*: BOOL;(*FPC下降抽屉到位传感器----------------------*)


(*EL1889-2*)
	X2_1 AT %I*: BOOL; (*送料上升到位光纤*)
	X2_2 AT %I*: BOOL; (*左送料上升到位光纤*)
	X2_3 AT %I*: BOOL; (*左收盘下降到位光纤*)
	X2_4 AT %I*: BOOL; (*右送盘上升到位光纤*)
	X2_5 AT %I*: BOOL;(*右收料下降到位光纤*)
	X2_6 AT %I*: BOOL;(*抽屉---------------*)
	X2_7 AT %I*: BOOL;(*撕膜电机吸膜负压表*)
	X2_8 AT %I*: BOOL;(*撕膜电机吸产品负压表*)
	X2_9 AT %I*: BOOL;(*TRAY盘抽屉上升到位传感器-----------------------*)
	X2_10 AT %I*: BOOL;(*左升降平移气缸SET*)
	X2_11 AT %I*: BOOL;(*左升降平移气缸RST*)
	X2_12 AT %I*: BOOL;(*左升降上下气缸SET*)
	X2_13 AT %I*: BOOL;(*左升降上下气缸RST*)
	X2_14 AT %I*: BOOL;(*左升降真空吸负压表*)
	X2_15 AT %I*: BOOL;(*TRAY盘抽屉下降到位传感器-----------------------*)
	X2_16 AT %I*: BOOL;(*滚压推入气缸SET*)

(*EL1889-3*)

	X3_1 AT %I*: BOOL;(*滚压推入气缸RST*)
	X3_2 AT %I*: BOOL;(*滚压上下气缸SET*)
	X3_3 AT %I*: BOOL;(*滚压上下气缸RST*)
	X3_4 AT %I*: BOOL;(*滚压翻转气缸SET*)
	X3_5 AT %I*: BOOL;(*滚压翻转气缸RST*)
	X3_6 AT %I*: BOOL;(*滚压平台真空吸负压表*)
	X3_7 AT %I*: BOOL;
	X3_8 AT %I*: BOOL;(*右升降平移气缸SET*)
	X3_9 AT %I*: BOOL;(*右升降平移气缸RST*)
	X3_10 AT %I*: BOOL;(*右升降上下气缸SET*)
	X3_11 AT %I*: BOOL;(*右升降上下气缸RST*)
	X3_12 AT %I*: BOOL;(*右升降真空吸负压表*)
	X3_13 AT %I*: BOOL;(*Pass-tray上料门感应--------------*)
	X3_14 AT %I*: BOOL;(*前门左门感应*)
	X3_15 AT %I*: BOOL;(*前门右门感应*)
	X3_16 AT %I*: BOOL;(*后门左门感应*)


(*EL1889-4*)

	X4_1 AT %I*: BOOL;(*后门右门感应*)
	X4_2 AT %I*: BOOL;(*HB上料门感应1*)
	X4_3 AT %I*: BOOL;(*HB上料门感应2*)
	X4_4 AT %I*: BOOL;(*启动按钮*)
	X4_5 AT %I*: BOOL;(*停止按钮*)
	X4_6 AT %I*: BOOL;(*复位按钮*)
	X4_7 AT %I*: BOOL;(*急停按钮*)
	X4_8 AT %I*: BOOL;(*轴11正极限*)
	X4_9 AT %I*: BOOL;(*轴11原点*)
	X4_10 AT %I*: BOOL;(*轴11反极限*)
	X4_11 AT %I*: BOOL;(*左移载上顶气缸SET1*)
	X4_12 AT %I*: BOOL;(*左移载上顶气缸Rst1*)
	X4_13 AT %I*: BOOL;(*左移载上顶气缸SET2*)
	X4_14 AT %I*: BOOL;(*左移载上顶气缸RST2*)
	X4_15 AT %I*: BOOL;
	X4_16 AT %I*: BOOL;


(*EL2889-0*)

	Y0_1 AT %Q*: BOOL; (*撕膜平台真空吸*)
	Y0_2 AT %Q*: BOOL; (*滑台2真空吸-------*)							(*滑台真空吸2222222222222*)
	Y0_3 AT %Q*: BOOL; (*撕膜电机吸料真空吸*)                                                 (*撕膜位置真空吸--------------*)
	Y0_4 AT %Q*: BOOL;(*矫正电机撕膜上气缸的夹子-----------------*)
	Y0_5 AT %Q*: BOOL; (*左载盘真空吸*)						(*滑台真空吸111111111111111111111*)
	Y0_6 AT %Q*: BOOL; (*左升降平移气缸*)
	Y0_7 AT %Q*: BOOL; (*左升降上下气缸*)
	Y0_8 AT %Q*: BOOL; (*左升降吸盘真空吸*)
	Y0_9 AT %Q*: BOOL;(*滚压滚轮气缸*)
	Y0_10 AT %Q*: BOOL; (*滚压推入气缸*)
	Y0_11 AT %Q*: BOOL; (*滚压下压压板气缸*)
	Y0_12 AT %Q*: BOOL; (*滚压平台真空吸*)
	Y0_13 AT %Q*: BOOL; (*滚压翻转气缸*)
	Y0_14 AT %Q*: BOOL; (*右载盘真空吸*)
	Y0_15 AT %Q*: BOOL;
	Y0_16 AT %Q*: BOOL; (*右升降平移气缸*)


(*EL2889-1*)

	Y1_1 AT %Q*: BOOL; (*右升降上下气缸*)
	Y1_2 AT %Q*: BOOL;(*右升降吸盘真空吸*)
	Y1_3 AT %Q*: BOOL;(*撕膜上顶气缸*)
	Y1_4 AT %Q*: BOOL;(*撕膜夹子撕膜上下气缸-----------------------*)
	Y1_5 AT %Q*: BOOL; (*门安全信号输出-到继电器-给机械手*)
	Y1_6 AT %Q*: BOOL;(*追加上顶气缸-------------------------------------------*)
	Y1_7 AT %Q*: BOOL;(*追加上顶气缸2-------------------------------------------*)
	Y1_8 AT %Q*: BOOL;
	Y1_9 AT %Q*: BOOL;(*FPC扣紧气缸*)
	Y1_10 AT %Q*: BOOL;(*初始----吹膜1*)
	Y1_11 AT %Q*: BOOL;(*吹膜2----------------*)
	Y1_12 AT %Q*: BOOL;
	Y1_13 AT %Q*: BOOL; (*绿灯*)
	Y1_14 AT %Q*: BOOL; (*黄灯*)
	Y1_15 AT %Q*: BOOL; (*红灯*)
	Y1_16 AT %Q*: BOOL; (*蜂鸣器*)

(*EL2889-1*)

	Y2_1 AT %Q*: BOOL;
	Y2_2 AT %Q*: BOOL;
	Y2_3 AT %Q*: BOOL;
	Y2_4 AT %Q*: BOOL;
	Y2_5 AT %Q*: BOOL;
	Y2_6 AT %Q*: BOOL;
	Y2_7 AT %Q*: BOOL;
	Y2_8 AT %Q*: BOOL;
	Y2_9 AT %Q*: BOOL;
	Y2_10 AT %Q*: BOOL;
	Y2_11 AT %Q*: BOOL;
	Y2_12 AT %Q*: BOOL;
	Y2_13 AT %Q*: BOOL;
	Y2_14 AT %Q*: BOOL;
	Y2_15 AT %Q*: BOOL;
	Y2_16 AT %Q*: BOOL;

END_VAR

(* Global variable list: Global_Variables_Special *)
VAR_GLOBAL

	Specila_Feed_FPC: BOOL;
	Specila_Feed_FPC_OFF: BOOL;



(*debug----------------视觉部分测试程序-------button*)
	Test_Camera_Run: BOOL;
	Test_Camera_Run1: BOOL;
(*气缸切换按钮*)
	BU1: BOOL;
	BU2: BOOL;

	Rset_Test1:BOOL;(*测试滑台1程序复位*)
	Rset_Test2:BOOL;(*测试滑台1程序复位*)

	Test_Camera_Run_loop: BOOL;
	Test_Camera_Run_loop1: BOOL;

	Rolling_Part_Run_Test:BOOL;
	Rolling_Part_Run_Test_OFF:BOOL;
	Rolling_Once_Run:BOOL;
	Rolling_Pushor_NOT:BOOL;

(*撕膜测试程序*)
	Film_Test:BOOL;
	Film_Test_OFF:BOOL;
	Film_Once_Run:BOOL;
	Qurensimo: BOOL;



END_VAR

(* Global variable list: TwinCAT_Configuration *)
(* Generated automatically by TwinCAT - (read only) *)
VAR_CONFIG
	.Axis1.PlcToNc AT %QB6 : PLCTONC_AXIS_REF;	(*  ~ {LinkedWith:TINC^NC-Task 1 SAF^Axes^Axis 1^Inputs^Axis 1_FromPlc} *)
	.Axis1.NcToPlc AT %IB10 : NCTOPLC_AXIS_REF;	(*  ~ {LinkedWith:TINC^NC-Task 1 SAF^Axes^Axis 1^Outputs^Axis 1_ToPlc} *)
	.Axis2.PlcToNc AT %QB134 : PLCTONC_AXIS_REF;	(*  ~ {LinkedWith:TINC^NC-Task 1 SAF^Axes^Axis 2^Inputs^Axis 2_FromPlc} *)
	.Axis2.NcToPlc AT %IB138 : NCTOPLC_AXIS_REF;	(*  ~ {LinkedWith:TINC^NC-Task 1 SAF^Axes^Axis 2^Outputs^Axis 2_ToPlc} *)
	.Axis3.PlcToNc AT %QB262 : PLCTONC_AXIS_REF;	(*  ~ {LinkedWith:TINC^NC-Task 1 SAF^Axes^Axis 3^Inputs^Axis 3_FromPlc} *)
	.Axis3.NcToPlc AT %IB266 : NCTOPLC_AXIS_REF;	(*  ~ {LinkedWith:TINC^NC-Task 1 SAF^Axes^Axis 3^Outputs^Axis 3_ToPlc} *)
	.Axis4.PlcToNc AT %QB390 : PLCTONC_AXIS_REF;	(*  ~ {LinkedWith:TINC^NC-Task 1 SAF^Axes^Axis 4^Inputs^Axis 4_FromPlc} *)
	.Axis4.NcToPlc AT %IB394 : NCTOPLC_AXIS_REF;	(*  ~ {LinkedWith:TINC^NC-Task 1 SAF^Axes^Axis 4^Outputs^Axis 4_ToPlc} *)
	.Axis5.PlcToNc AT %QB518 : PLCTONC_AXIS_REF;	(*  ~ {LinkedWith:TINC^NC-Task 1 SAF^Axes^Axis 5^Inputs^Axis 5_FromPlc} *)
	.Axis5.NcToPlc AT %IB522 : NCTOPLC_AXIS_REF;	(*  ~ {LinkedWith:TINC^NC-Task 1 SAF^Axes^Axis 5^Outputs^Axis 5_ToPlc} *)
	.Axis6.PlcToNc AT %QB646 : PLCTONC_AXIS_REF;	(*  ~ {LinkedWith:TINC^NC-Task 1 SAF^Axes^Axis 6^Inputs^Axis 6_FromPlc} *)
	.Axis6.NcToPlc AT %IB650 : NCTOPLC_AXIS_REF;	(*  ~ {LinkedWith:TINC^NC-Task 1 SAF^Axes^Axis 6^Outputs^Axis 6_ToPlc} *)
	.Axis7.PlcToNc AT %QB774 : PLCTONC_AXIS_REF;	(*  ~ {LinkedWith:TINC^NC-Task 1 SAF^Axes^Axis 7^Inputs^Axis 7_FromPlc} *)
	.Axis7.NcToPlc AT %IB778 : NCTOPLC_AXIS_REF;	(*  ~ {LinkedWith:TINC^NC-Task 1 SAF^Axes^Axis 7^Outputs^Axis 7_ToPlc} *)
	.Axis8.PlcToNc AT %QB902 : PLCTONC_AXIS_REF;	(*  ~ {LinkedWith:TINC^NC-Task 1 SAF^Axes^Axis 8^Inputs^Axis 8_FromPlc} *)
	.Axis8.NcToPlc AT %IB906 : NCTOPLC_AXIS_REF;	(*  ~ {LinkedWith:TINC^NC-Task 1 SAF^Axes^Axis 8^Outputs^Axis 8_ToPlc} *)
	.Axis9.PlcToNc AT %QB1030 : PLCTONC_AXIS_REF;	(*  ~ {LinkedWith:TINC^NC-Task 1 SAF^Axes^Axis 9^Inputs^Axis 9_FromPlc} *)
	.Axis9.NcToPlc AT %IB1034 : NCTOPLC_AXIS_REF;	(*  ~ {LinkedWith:TINC^NC-Task 1 SAF^Axes^Axis 9^Outputs^Axis 9_ToPlc} *)
	.Axis10.PlcToNc AT %QB1158 : PLCTONC_AXIS_REF;	(*  ~ {LinkedWith:TINC^NC-Task 1 SAF^Axes^Axis 10^Inputs^Axis 10_FromPlc} *)
	.Axis10.NcToPlc AT %IB1162 : NCTOPLC_AXIS_REF;	(*  ~ {LinkedWith:TINC^NC-Task 1 SAF^Axes^Axis 10^Outputs^Axis 10_ToPlc} *)
	.Axis11.PlcToNc AT %QB1286 : PLCTONC_AXIS_REF;	(*  ~ {LinkedWith:TINC^NC-Task 1 SAF^Axes^Axis 11^Inputs^Axis 11_FromPlc} *)
	.Axis11.NcToPlc AT %IB1290 : NCTOPLC_AXIS_REF;	(*  ~ {LinkedWith:TINC^NC-Task 1 SAF^Axes^Axis 11^Outputs^Axis 11_ToPlc} *)
	.Axis13.PlcToNc AT %QB1416 : PLCTONC_AXIS_REF;
	.Axis13.NcToPlc AT %IB1422 : NCTOPLC_AXIS_REF;
	.Axis12.PlcToNc AT %QB1544 : PLCTONC_AXIS_REF;
	.Axis12.NcToPlc AT %IB1550 : NCTOPLC_AXIS_REF;
	.F_push AT %IB1420 : INT;
	.X0_1 AT %IX0.0 : BOOL;	(*  ~ {LinkedWith:TIID^Device 3 (EtherCAT)^Term 1 (EK1100)^Term 2 (EL1889)^Channel 1^Input} *)
	.X0_2 AT %IX0.1 : BOOL;	(*  ~ {LinkedWith:TIID^Device 3 (EtherCAT)^Term 1 (EK1100)^Term 2 (EL1889)^Channel 2^Input} *)
	.X0_3 AT %IX0.2 : BOOL;	(*  ~ {LinkedWith:TIID^Device 3 (EtherCAT)^Term 1 (EK1100)^Term 2 (EL1889)^Channel 3^Input} *)
	.X0_4 AT %IX0.3 : BOOL;	(*  ~ {LinkedWith:TIID^Device 3 (EtherCAT)^Term 1 (EK1100)^Term 2 (EL1889)^Channel 4^Input} *)
	.X0_5 AT %IX0.4 : BOOL;	(*  ~ {LinkedWith:TIID^Device 3 (EtherCAT)^Term 1 (EK1100)^Term 2 (EL1889)^Channel 5^Input} *)
	.X0_6 AT %IX0.5 : BOOL;	(*  ~ {LinkedWith:TIID^Device 3 (EtherCAT)^Term 1 (EK1100)^Term 2 (EL1889)^Channel 6^Input} *)
	.X0_7 AT %IX0.6 : BOOL;	(*  ~ {LinkedWith:TIID^Device 3 (EtherCAT)^Term 1 (EK1100)^Term 2 (EL1889)^Channel 7^Input} *)
	.X0_8 AT %IX0.7 : BOOL;	(*  ~ {LinkedWith:TIID^Device 3 (EtherCAT)^Term 1 (EK1100)^Term 2 (EL1889)^Channel 8^Input} *)
	.X0_9 AT %IX1.0 : BOOL;	(*  ~ {LinkedWith:TIID^Device 3 (EtherCAT)^Term 1 (EK1100)^Term 2 (EL1889)^Channel 9^Input} *)
	.X0_10 AT %IX1.1 : BOOL;	(*  ~ {LinkedWith:TIID^Device 3 (EtherCAT)^Term 1 (EK1100)^Term 2 (EL1889)^Channel 10^Input} *)
	.X0_11 AT %IX1.2 : BOOL;	(*  ~ {LinkedWith:TIID^Device 3 (EtherCAT)^Term 1 (EK1100)^Term 2 (EL1889)^Channel 11^Input} *)
	.X0_12 AT %IX1.3 : BOOL;	(*  ~ {LinkedWith:TIID^Device 3 (EtherCAT)^Term 1 (EK1100)^Term 2 (EL1889)^Channel 12^Input} *)
	.X0_13 AT %IX1.4 : BOOL;	(*  ~ {LinkedWith:TIID^Device 3 (EtherCAT)^Term 1 (EK1100)^Term 2 (EL1889)^Channel 13^Input} *)
	.X0_14 AT %IX1.5 : BOOL;	(*  ~ {LinkedWith:TIID^Device 3 (EtherCAT)^Term 1 (EK1100)^Term 2 (EL1889)^Channel 14^Input} *)
	.X0_15 AT %IX1.6 : BOOL;	(*  ~ {LinkedWith:TIID^Device 3 (EtherCAT)^Term 1 (EK1100)^Term 2 (EL1889)^Channel 15^Input} *)
	.X0_16 AT %IX1.7 : BOOL;	(*  ~ {LinkedWith:TIID^Device 3 (EtherCAT)^Term 1 (EK1100)^Term 2 (EL1889)^Channel 16^Input} *)
	.X1_1 AT %IX2.0 : BOOL;	(*  ~ {LinkedWith:TIID^Device 3 (EtherCAT)^Term 1 (EK1100)^Term 3 (EL1889)^Channel 1^Input} *)
	.X1_2 AT %IX2.1 : BOOL;	(*  ~ {LinkedWith:TIID^Device 3 (EtherCAT)^Term 1 (EK1100)^Term 3 (EL1889)^Channel 2^Input} *)
	.X1_3 AT %IX2.2 : BOOL;	(*  ~ {LinkedWith:TIID^Device 3 (EtherCAT)^Term 1 (EK1100)^Term 3 (EL1889)^Channel 3^Input} *)
	.X1_4 AT %IX2.3 : BOOL;	(*  ~ {LinkedWith:TIID^Device 3 (EtherCAT)^Term 1 (EK1100)^Term 3 (EL1889)^Channel 4^Input} *)
	.X1_5 AT %IX2.4 : BOOL;	(*  ~ {LinkedWith:TIID^Device 3 (EtherCAT)^Term 1 (EK1100)^Term 3 (EL1889)^Channel 5^Input} *)
	.X1_6 AT %IX2.5 : BOOL;	(*  ~ {LinkedWith:TIID^Device 3 (EtherCAT)^Term 1 (EK1100)^Term 3 (EL1889)^Channel 6^Input} *)
	.X1_7 AT %IX2.6 : BOOL;	(*  ~ {LinkedWith:TIID^Device 3 (EtherCAT)^Term 1 (EK1100)^Term 3 (EL1889)^Channel 7^Input} *)
	.X1_8 AT %IX2.7 : BOOL;	(*  ~ {LinkedWith:TIID^Device 3 (EtherCAT)^Term 1 (EK1100)^Term 3 (EL1889)^Channel 8^Input} *)
	.X1_9 AT %IX3.0 : BOOL;	(*  ~ {LinkedWith:TIID^Device 3 (EtherCAT)^Term 1 (EK1100)^Term 3 (EL1889)^Channel 9^Input} *)
	.X1_10 AT %IX3.1 : BOOL;	(*  ~ {LinkedWith:TIID^Device 3 (EtherCAT)^Term 1 (EK1100)^Term 3 (EL1889)^Channel 10^Input} *)
	.X1_11 AT %IX3.2 : BOOL;	(*  ~ {LinkedWith:TIID^Device 3 (EtherCAT)^Term 1 (EK1100)^Term 3 (EL1889)^Channel 11^Input} *)
	.X1_12 AT %IX3.3 : BOOL;	(*  ~ {LinkedWith:TIID^Device 3 (EtherCAT)^Term 1 (EK1100)^Term 3 (EL1889)^Channel 12^Input} *)
	.X1_13 AT %IX3.4 : BOOL;	(*  ~ {LinkedWith:TIID^Device 3 (EtherCAT)^Term 1 (EK1100)^Term 3 (EL1889)^Channel 13^Input} *)
	.X1_14 AT %IX3.5 : BOOL;	(*  ~ {LinkedWith:TIID^Device 3 (EtherCAT)^Term 1 (EK1100)^Term 3 (EL1889)^Channel 14^Input} *)
	.X1_15 AT %IX3.6 : BOOL;	(*  ~ {LinkedWith:TIID^Device 3 (EtherCAT)^Term 1 (EK1100)^Term 3 (EL1889)^Channel 15^Input} *)
	.X1_16 AT %IX3.7 : BOOL;	(*  ~ {LinkedWith:TIID^Device 3 (EtherCAT)^Term 1 (EK1100)^Term 3 (EL1889)^Channel 16^Input} *)
	.X2_1 AT %IX4.0 : BOOL;	(*  ~ {LinkedWith:TIID^Device 3 (EtherCAT)^Term 1 (EK1100)^Term 4 (EL1889)^Channel 1^Input} *)
	.X2_2 AT %IX4.1 : BOOL;	(*  ~ {LinkedWith:TIID^Device 3 (EtherCAT)^Term 1 (EK1100)^Term 4 (EL1889)^Channel 2^Input} *)
	.X2_3 AT %IX4.2 : BOOL;	(*  ~ {LinkedWith:TIID^Device 3 (EtherCAT)^Term 1 (EK1100)^Term 4 (EL1889)^Channel 3^Input} *)
	.X2_4 AT %IX4.3 : BOOL;	(*  ~ {LinkedWith:TIID^Device 3 (EtherCAT)^Term 1 (EK1100)^Term 4 (EL1889)^Channel 4^Input} *)
	.X2_5 AT %IX4.4 : BOOL;	(*  ~ {LinkedWith:TIID^Device 3 (EtherCAT)^Term 1 (EK1100)^Term 4 (EL1889)^Channel 5^Input} *)
	.X2_6 AT %IX4.5 : BOOL;	(*  ~ {LinkedWith:TIID^Device 3 (EtherCAT)^Term 1 (EK1100)^Term 4 (EL1889)^Channel 6^Input} *)
	.X2_7 AT %IX4.6 : BOOL;	(*  ~ {LinkedWith:TIID^Device 3 (EtherCAT)^Term 1 (EK1100)^Term 4 (EL1889)^Channel 7^Input} *)
	.X2_8 AT %IX4.7 : BOOL;	(*  ~ {LinkedWith:TIID^Device 3 (EtherCAT)^Term 1 (EK1100)^Term 4 (EL1889)^Channel 8^Input} *)
	.X2_9 AT %IX5.0 : BOOL;	(*  ~ {LinkedWith:TIID^Device 3 (EtherCAT)^Term 1 (EK1100)^Term 4 (EL1889)^Channel 9^Input} *)
	.X2_10 AT %IX5.1 : BOOL;	(*  ~ {LinkedWith:TIID^Device 3 (EtherCAT)^Term 1 (EK1100)^Term 4 (EL1889)^Channel 10^Input} *)
	.X2_11 AT %IX5.2 : BOOL;	(*  ~ {LinkedWith:TIID^Device 3 (EtherCAT)^Term 1 (EK1100)^Term 4 (EL1889)^Channel 11^Input} *)
	.X2_12 AT %IX5.3 : BOOL;	(*  ~ {LinkedWith:TIID^Device 3 (EtherCAT)^Term 1 (EK1100)^Term 4 (EL1889)^Channel 12^Input} *)
	.X2_13 AT %IX5.4 : BOOL;	(*  ~ {LinkedWith:TIID^Device 3 (EtherCAT)^Term 1 (EK1100)^Term 4 (EL1889)^Channel 13^Input} *)
	.X2_14 AT %IX5.5 : BOOL;	(*  ~ {LinkedWith:TIID^Device 3 (EtherCAT)^Term 1 (EK1100)^Term 4 (EL1889)^Channel 14^Input} *)
	.X2_15 AT %IX5.6 : BOOL;	(*  ~ {LinkedWith:TIID^Device 3 (EtherCAT)^Term 1 (EK1100)^Term 4 (EL1889)^Channel 15^Input} *)
	.X2_16 AT %IX5.7 : BOOL;	(*  ~ {LinkedWith:TIID^Device 3 (EtherCAT)^Term 1 (EK1100)^Term 4 (EL1889)^Channel 16^Input} *)
	.X3_1 AT %IX6.0 : BOOL;	(*  ~ {LinkedWith:TIID^Device 3 (EtherCAT)^Term 1 (EK1100)^Term 5 (EL1889)^Channel 1^Input} *)
	.X3_2 AT %IX6.1 : BOOL;	(*  ~ {LinkedWith:TIID^Device 3 (EtherCAT)^Term 1 (EK1100)^Term 5 (EL1889)^Channel 2^Input} *)
	.X3_3 AT %IX6.2 : BOOL;	(*  ~ {LinkedWith:TIID^Device 3 (EtherCAT)^Term 1 (EK1100)^Term 5 (EL1889)^Channel 3^Input} *)
	.X3_4 AT %IX6.3 : BOOL;	(*  ~ {LinkedWith:TIID^Device 3 (EtherCAT)^Term 1 (EK1100)^Term 5 (EL1889)^Channel 4^Input} *)
	.X3_5 AT %IX6.4 : BOOL;	(*  ~ {LinkedWith:TIID^Device 3 (EtherCAT)^Term 1 (EK1100)^Term 5 (EL1889)^Channel 5^Input} *)
	.X3_6 AT %IX6.5 : BOOL;	(*  ~ {LinkedWith:TIID^Device 3 (EtherCAT)^Term 1 (EK1100)^Term 5 (EL1889)^Channel 6^Input} *)
	.X3_7 AT %IX6.6 : BOOL;	(*  ~ {LinkedWith:TIID^Device 3 (EtherCAT)^Term 1 (EK1100)^Term 5 (EL1889)^Channel 7^Input} *)
	.X3_8 AT %IX6.7 : BOOL;	(*  ~ {LinkedWith:TIID^Device 3 (EtherCAT)^Term 1 (EK1100)^Term 5 (EL1889)^Channel 8^Input} *)
	.X3_9 AT %IX7.0 : BOOL;	(*  ~ {LinkedWith:TIID^Device 3 (EtherCAT)^Term 1 (EK1100)^Term 5 (EL1889)^Channel 9^Input} *)
	.X3_10 AT %IX7.1 : BOOL;	(*  ~ {LinkedWith:TIID^Device 3 (EtherCAT)^Term 1 (EK1100)^Term 5 (EL1889)^Channel 10^Input} *)
	.X3_11 AT %IX7.2 : BOOL;	(*  ~ {LinkedWith:TIID^Device 3 (EtherCAT)^Term 1 (EK1100)^Term 5 (EL1889)^Channel 11^Input} *)
	.X3_12 AT %IX7.3 : BOOL;	(*  ~ {LinkedWith:TIID^Device 3 (EtherCAT)^Term 1 (EK1100)^Term 5 (EL1889)^Channel 12^Input} *)
	.X3_13 AT %IX7.4 : BOOL;	(*  ~ {LinkedWith:TIID^Device 3 (EtherCAT)^Term 1 (EK1100)^Term 5 (EL1889)^Channel 13^Input} *)
	.X3_14 AT %IX7.5 : BOOL;	(*  ~ {LinkedWith:TIID^Device 3 (EtherCAT)^Term 1 (EK1100)^Term 5 (EL1889)^Channel 14^Input} *)
	.X3_15 AT %IX7.6 : BOOL;	(*  ~ {LinkedWith:TIID^Device 3 (EtherCAT)^Term 1 (EK1100)^Term 5 (EL1889)^Channel 15^Input} *)
	.X3_16 AT %IX7.7 : BOOL;	(*  ~ {LinkedWith:TIID^Device 3 (EtherCAT)^Term 1 (EK1100)^Term 5 (EL1889)^Channel 16^Input} *)
	.X4_1 AT %IX8.0 : BOOL;	(*  ~ {LinkedWith:TIID^Device 3 (EtherCAT)^Term 1 (EK1100)^Term 6 (EL1889)^Channel 1^Input} *)
	.X4_2 AT %IX8.1 : BOOL;	(*  ~ {LinkedWith:TIID^Device 3 (EtherCAT)^Term 1 (EK1100)^Term 6 (EL1889)^Channel 2^Input} *)
	.X4_3 AT %IX8.2 : BOOL;	(*  ~ {LinkedWith:TIID^Device 3 (EtherCAT)^Term 1 (EK1100)^Term 6 (EL1889)^Channel 3^Input} *)
	.X4_4 AT %IX8.3 : BOOL;	(*  ~ {LinkedWith:TIID^Device 3 (EtherCAT)^Term 1 (EK1100)^Term 6 (EL1889)^Channel 4^Input} *)
	.X4_5 AT %IX8.4 : BOOL;	(*  ~ {LinkedWith:TIID^Device 3 (EtherCAT)^Term 1 (EK1100)^Term 6 (EL1889)^Channel 5^Input} *)
	.X4_6 AT %IX8.5 : BOOL;	(*  ~ {LinkedWith:TIID^Device 3 (EtherCAT)^Term 1 (EK1100)^Term 6 (EL1889)^Channel 6^Input} *)
	.X4_7 AT %IX8.6 : BOOL;	(*  ~ {LinkedWith:TIID^Device 3 (EtherCAT)^Term 1 (EK1100)^Term 6 (EL1889)^Channel 7^Input} *)
	.X4_8 AT %IX8.7 : BOOL;	(*  ~ {LinkedWith:TIID^Device 3 (EtherCAT)^Term 1 (EK1100)^Term 6 (EL1889)^Channel 8^Input} *)
	.X4_9 AT %IX9.0 : BOOL;	(*  ~ {LinkedWith:TIID^Device 3 (EtherCAT)^Term 1 (EK1100)^Term 6 (EL1889)^Channel 9^Input} *)
	.X4_10 AT %IX9.1 : BOOL;	(*  ~ {LinkedWith:TIID^Device 3 (EtherCAT)^Term 1 (EK1100)^Term 6 (EL1889)^Channel 10^Input} *)
	.X4_11 AT %IX9.2 : BOOL;	(*  ~ {LinkedWith:TIID^Device 3 (EtherCAT)^Term 1 (EK1100)^Term 6 (EL1889)^Channel 11^Input} *)
	.X4_12 AT %IX9.3 : BOOL;	(*  ~ {LinkedWith:TIID^Device 3 (EtherCAT)^Term 1 (EK1100)^Term 6 (EL1889)^Channel 12^Input} *)
	.X4_13 AT %IX9.4 : BOOL;	(*  ~ {LinkedWith:TIID^Device 3 (EtherCAT)^Term 1 (EK1100)^Term 6 (EL1889)^Channel 13^Input} *)
	.X4_14 AT %IX9.5 : BOOL;	(*  ~ {LinkedWith:TIID^Device 3 (EtherCAT)^Term 1 (EK1100)^Term 6 (EL1889)^Channel 14^Input} *)
	.X4_15 AT %IX9.6 : BOOL;	(*  ~ {LinkedWith:TIID^Device 3 (EtherCAT)^Term 1 (EK1100)^Term 6 (EL1889)^Channel 15^Input} *)
	.X4_16 AT %IX9.7 : BOOL;	(*  ~ {LinkedWith:TIID^Device 3 (EtherCAT)^Term 1 (EK1100)^Term 6 (EL1889)^Channel 16^Input} *)
	.Y0_1 AT %QX0.0 : BOOL;	(*  ~ {LinkedWith:TIID^Device 3 (EtherCAT)^Term 1 (EK1100)^Term 7 (EL2889)^Channel 1^Output} *)
	.Y0_2 AT %QX0.1 : BOOL;	(*  ~ {LinkedWith:TIID^Device 3 (EtherCAT)^Term 1 (EK1100)^Term 7 (EL2889)^Channel 2^Output} *)
	.Y0_3 AT %QX0.2 : BOOL;	(*  ~ {LinkedWith:TIID^Device 3 (EtherCAT)^Term 1 (EK1100)^Term 7 (EL2889)^Channel 3^Output} *)
	.Y0_4 AT %QX0.3 : BOOL;	(*  ~ {LinkedWith:TIID^Device 3 (EtherCAT)^Term 1 (EK1100)^Term 7 (EL2889)^Channel 4^Output} *)
	.Y0_5 AT %QX0.4 : BOOL;	(*  ~ {LinkedWith:TIID^Device 3 (EtherCAT)^Term 1 (EK1100)^Term 7 (EL2889)^Channel 5^Output} *)
	.Y0_6 AT %QX0.5 : BOOL;	(*  ~ {LinkedWith:TIID^Device 3 (EtherCAT)^Term 1 (EK1100)^Term 7 (EL2889)^Channel 6^Output} *)
	.Y0_7 AT %QX0.6 : BOOL;	(*  ~ {LinkedWith:TIID^Device 3 (EtherCAT)^Term 1 (EK1100)^Term 7 (EL2889)^Channel 7^Output} *)
	.Y0_8 AT %QX0.7 : BOOL;	(*  ~ {LinkedWith:TIID^Device 3 (EtherCAT)^Term 1 (EK1100)^Term 7 (EL2889)^Channel 8^Output} *)
	.Y0_9 AT %QX1.0 : BOOL;	(*  ~ {LinkedWith:TIID^Device 3 (EtherCAT)^Term 1 (EK1100)^Term 7 (EL2889)^Channel 9^Output} *)
	.Y0_10 AT %QX1.1 : BOOL;	(*  ~ {LinkedWith:TIID^Device 3 (EtherCAT)^Term 1 (EK1100)^Term 7 (EL2889)^Channel 10^Output} *)
	.Y0_11 AT %QX1.2 : BOOL;	(*  ~ {LinkedWith:TIID^Device 3 (EtherCAT)^Term 1 (EK1100)^Term 7 (EL2889)^Channel 11^Output} *)
	.Y0_12 AT %QX1.3 : BOOL;	(*  ~ {LinkedWith:TIID^Device 3 (EtherCAT)^Term 1 (EK1100)^Term 7 (EL2889)^Channel 12^Output} *)
	.Y0_13 AT %QX1.4 : BOOL;	(*  ~ {LinkedWith:TIID^Device 3 (EtherCAT)^Term 1 (EK1100)^Term 7 (EL2889)^Channel 13^Output} *)
	.Y0_14 AT %QX1.5 : BOOL;	(*  ~ {LinkedWith:TIID^Device 3 (EtherCAT)^Term 1 (EK1100)^Term 7 (EL2889)^Channel 14^Output} *)
	.Y0_15 AT %QX1.6 : BOOL;	(*  ~ {LinkedWith:TIID^Device 3 (EtherCAT)^Term 1 (EK1100)^Term 7 (EL2889)^Channel 15^Output} *)
	.Y0_16 AT %QX1.7 : BOOL;	(*  ~ {LinkedWith:TIID^Device 3 (EtherCAT)^Term 1 (EK1100)^Term 7 (EL2889)^Channel 16^Output} *)
	.Y1_1 AT %QX2.0 : BOOL;	(*  ~ {LinkedWith:TIID^Device 3 (EtherCAT)^Term 1 (EK1100)^Term 8 (EL2889)^Channel 1^Output} *)
	.Y1_2 AT %QX2.1 : BOOL;	(*  ~ {LinkedWith:TIID^Device 3 (EtherCAT)^Term 1 (EK1100)^Term 8 (EL2889)^Channel 2^Output} *)
	.Y1_3 AT %QX2.2 : BOOL;	(*  ~ {LinkedWith:TIID^Device 3 (EtherCAT)^Term 1 (EK1100)^Term 8 (EL2889)^Channel 3^Output} *)
	.Y1_4 AT %QX2.3 : BOOL;	(*  ~ {LinkedWith:TIID^Device 3 (EtherCAT)^Term 1 (EK1100)^Term 8 (EL2889)^Channel 4^Output} *)
	.Y1_5 AT %QX2.4 : BOOL;	(*  ~ {LinkedWith:TIID^Device 3 (EtherCAT)^Term 1 (EK1100)^Term 8 (EL2889)^Channel 5^Output} *)
	.Y1_6 AT %QX2.5 : BOOL;	(*  ~ {LinkedWith:TIID^Device 3 (EtherCAT)^Term 1 (EK1100)^Term 8 (EL2889)^Channel 6^Output} *)
	.Y1_7 AT %QX2.6 : BOOL;	(*  ~ {LinkedWith:TIID^Device 3 (EtherCAT)^Term 1 (EK1100)^Term 8 (EL2889)^Channel 7^Output} *)
	.Y1_8 AT %QX2.7 : BOOL;	(*  ~ {LinkedWith:TIID^Device 3 (EtherCAT)^Term 1 (EK1100)^Term 8 (EL2889)^Channel 8^Output} *)
	.Y1_9 AT %QX3.0 : BOOL;	(*  ~ {LinkedWith:TIID^Device 3 (EtherCAT)^Term 1 (EK1100)^Term 8 (EL2889)^Channel 9^Output} *)
	.Y1_10 AT %QX3.1 : BOOL;	(*  ~ {LinkedWith:TIID^Device 3 (EtherCAT)^Term 1 (EK1100)^Term 8 (EL2889)^Channel 10^Output} *)
	.Y1_11 AT %QX3.2 : BOOL;	(*  ~ {LinkedWith:TIID^Device 3 (EtherCAT)^Term 1 (EK1100)^Term 8 (EL2889)^Channel 11^Output} *)
	.Y1_12 AT %QX3.3 : BOOL;	(*  ~ {LinkedWith:TIID^Device 3 (EtherCAT)^Term 1 (EK1100)^Term 8 (EL2889)^Channel 12^Output} *)
	.Y1_13 AT %QX3.4 : BOOL;	(*  ~ {LinkedWith:TIID^Device 3 (EtherCAT)^Term 1 (EK1100)^Term 8 (EL2889)^Channel 13^Output} *)
	.Y1_14 AT %QX3.5 : BOOL;	(*  ~ {LinkedWith:TIID^Device 3 (EtherCAT)^Term 1 (EK1100)^Term 8 (EL2889)^Channel 14^Output} *)
	.Y1_15 AT %QX3.6 : BOOL;	(*  ~ {LinkedWith:TIID^Device 3 (EtherCAT)^Term 1 (EK1100)^Term 8 (EL2889)^Channel 15^Output} *)
	.Y1_16 AT %QX3.7 : BOOL;	(*  ~ {LinkedWith:TIID^Device 3 (EtherCAT)^Term 1 (EK1100)^Term 8 (EL2889)^Channel 16^Output} *)
	.Y2_1 AT %QX4.0 : BOOL;	(*  ~ {LinkedWith:TIID^Device 3 (EtherCAT)^Term 1 (EK1100)^Term 9 (EL2889)^Channel 1^Output} *)
	.Y2_2 AT %QX4.1 : BOOL;	(*  ~ {LinkedWith:TIID^Device 3 (EtherCAT)^Term 1 (EK1100)^Term 9 (EL2889)^Channel 2^Output} *)
	.Y2_3 AT %QX4.2 : BOOL;	(*  ~ {LinkedWith:TIID^Device 3 (EtherCAT)^Term 1 (EK1100)^Term 9 (EL2889)^Channel 3^Output} *)
	.Y2_4 AT %QX4.3 : BOOL;	(*  ~ {LinkedWith:TIID^Device 3 (EtherCAT)^Term 1 (EK1100)^Term 9 (EL2889)^Channel 4^Output} *)
	.Y2_5 AT %QX4.4 : BOOL;	(*  ~ {LinkedWith:TIID^Device 3 (EtherCAT)^Term 1 (EK1100)^Term 9 (EL2889)^Channel 5^Output} *)
	.Y2_6 AT %QX4.5 : BOOL;	(*  ~ {LinkedWith:TIID^Device 3 (EtherCAT)^Term 1 (EK1100)^Term 9 (EL2889)^Channel 6^Output} *)
	.Y2_7 AT %QX4.6 : BOOL;	(*  ~ {LinkedWith:TIID^Device 3 (EtherCAT)^Term 1 (EK1100)^Term 9 (EL2889)^Channel 7^Output} *)
	.Y2_8 AT %QX4.7 : BOOL;	(*  ~ {LinkedWith:TIID^Device 3 (EtherCAT)^Term 1 (EK1100)^Term 9 (EL2889)^Channel 8^Output} *)
	.Y2_9 AT %QX5.0 : BOOL;	(*  ~ {LinkedWith:TIID^Device 3 (EtherCAT)^Term 1 (EK1100)^Term 9 (EL2889)^Channel 9^Output} *)
	.Y2_10 AT %QX5.1 : BOOL;	(*  ~ {LinkedWith:TIID^Device 3 (EtherCAT)^Term 1 (EK1100)^Term 9 (EL2889)^Channel 10^Output} *)
	.Y2_11 AT %QX5.2 : BOOL;	(*  ~ {LinkedWith:TIID^Device 3 (EtherCAT)^Term 1 (EK1100)^Term 9 (EL2889)^Channel 11^Output} *)
	.Y2_12 AT %QX5.3 : BOOL;	(*  ~ {LinkedWith:TIID^Device 3 (EtherCAT)^Term 1 (EK1100)^Term 9 (EL2889)^Channel 12^Output} *)
	.Y2_13 AT %QX5.4 : BOOL;	(*  ~ {LinkedWith:TIID^Device 3 (EtherCAT)^Term 1 (EK1100)^Term 9 (EL2889)^Channel 13^Output} *)
	.Y2_14 AT %QX5.5 : BOOL;	(*  ~ {LinkedWith:TIID^Device 3 (EtherCAT)^Term 1 (EK1100)^Term 9 (EL2889)^Channel 14^Output} *)
	.Y2_15 AT %QX5.6 : BOOL;	(*  ~ {LinkedWith:TIID^Device 3 (EtherCAT)^Term 1 (EK1100)^Term 9 (EL2889)^Channel 15^Output} *)
	.Y2_16 AT %QX5.7 : BOOL;	(*  ~ {LinkedWith:TIID^Device 3 (EtherCAT)^Term 1 (EK1100)^Term 9 (EL2889)^Channel 16^Output} *)
END_VAR

(* POU MAIN, ST *)
PROGRAM MAIN
VAR
END_VAR
RollTime :=(A10_w1-A10_w2)/D20_1;

(*电机功能块*)
Home_Pro();Power_Pro();Abs_Pro();Halt_Pro();Motion_Rst();MotionRst_Pro();PTF_Pro();Axis_Status_Check();
Axis_Status();Limit_Mapping();Speed_Setting();

(*调试模式*)
Axis1_Debug_Model();Axis2_Debug_Model();Axis3_Debug_Model();Axis4_Debug_Model();Axis5_Debug_Model();
Axis6_Debug_Model();Axis7_Debug_Model();Axis8_Debug_Model();Axis9_Debug_Model();Axis10_Debug_Model();
Axis11_Debug_Model();
Others_Debug_Model();
Debug12();


Feed_alam_status();
(*回原点*)
Axis1_Home_Back();Axis2_Home_Back();Axis3_Home_Back();Axis4_Home_Back();Axis5_Home_Back();
Axis6_Home_Back();Axis7_Home_Back();Axis8_Home_Back();Axis9_Home_Back();Axis10_Home_Back();
Axis11_Home_Back();
Home_Ptf_Rst();
(*报警，暂停，急停*)
Alarm_Monitoring();
Message_And_Status();
Pause();
Emergency_Stop();
Lamp();
Coord_Test();
Y09LOOP();



Camera_Test();Camera_Test_1();Camera_Test_loop();Camera_Test_loop_1();
Rolling_Part_1();


New_IniRun(bstart1:=X4_4 OR All_Start , bhold1:=Total_Pause , breset1:= );


Film_Handel_Pro_1(bstart1:=X4_4 OR All_Start , bhold1:=Total_Pause , breset1:= );

Right_Translation(bstart1:=X4_4 OR All_Start , bhold1:=Total_Pause , breset1:= );
Rolling_Part(bstart1:=X4_4 OR All_Start , bhold1:=Total_Pause , breset1:= );

Left_Carry(bstart1:=X4_4 OR All_Start , bhold1:=Total_Pause , breset1:= );


Liftin_Feed_1(bstart1:=X4_4 OR All_Start , bhold1:=Total_Pause , breset1:= );

Liftin_Feed_Left_1(bstart1:=X4_4 OR All_Start , bhold1:=Total_Pause , breset1:= );


Liftin_Feed_Left_2(bstart1:=X4_4 OR All_Start , bhold1:=Total_Pause , breset1:= );


New_Table_1(bstart1:=X4_4 OR All_Start , bhold1:=Total_Pause , breset1:= );
New_Table_2(bstart1:=X4_4 OR All_Start , bhold1:=Total_Pause , breset1:= );
Film_Test1();

Rool_Test();

Liftin_Feed_Right_Down(bstart1:=X4_4 OR All_Start , bhold1:=Total_Pause , breset1:= );
Liftin_Feed_Right_Up(bstart1:=X4_4 OR All_Start , bhold1:=Total_Pause , breset1:= );
Right_Carry_1(bstart1:=X4_4 OR All_Start , bhold1:=Total_Pause , breset1:= );
PID2();
PID1();

(*Rolling_Part_Just(bstart1:=X4_4 OR All_Start , bhold1:=Total_Pause , breset1:= );*)

(*New_Table_3(bstart1:=X4_4 OR All_Start , bhold1:=Total_Pause , breset1:= );*)
END_PROGRAM

(* POU Other_Folder/Motion/Home_Pro, FBD *)
PROGRAM Home_Pro
VAR
END_VAR
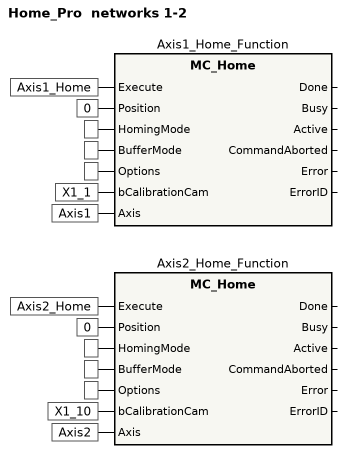
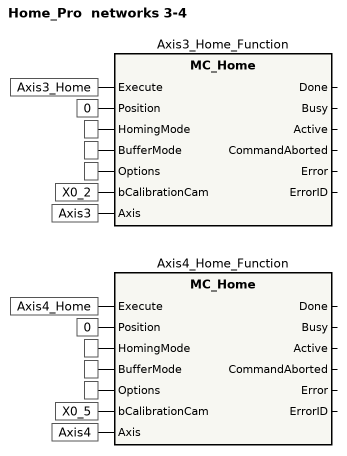
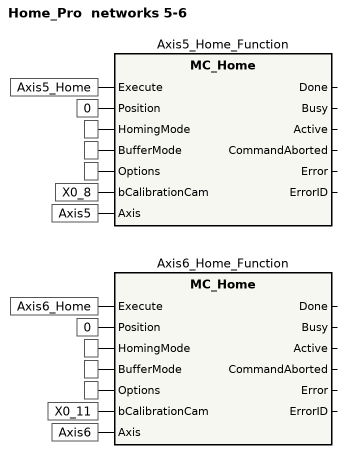
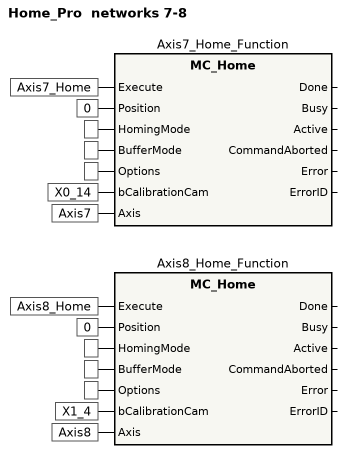
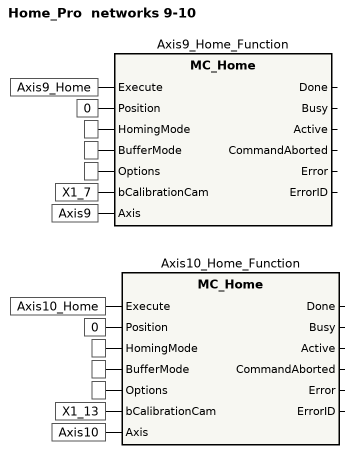
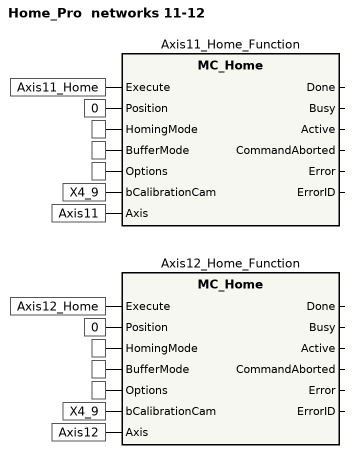
_FBD_ (* Function Block Diagram *)
NETWORK 1
	Axis1_Home_Function:MC_Home(Execute: Axis1_Home, Position: 0, HomingMode: , BufferMode: , Options: , bCalibrationCam: X1_1, Axis: Axis1)
NETWORK 2
	Axis2_Home_Function:MC_Home(Execute: Axis2_Home, Position: 0, HomingMode: , BufferMode: , Options: , bCalibrationCam: X1_10, Axis: Axis2)
NETWORK 3
	Axis3_Home_Function:MC_Home(Execute: Axis3_Home, Position: 0, HomingMode: , BufferMode: , Options: , bCalibrationCam: X0_2, Axis: Axis3)
NETWORK 4
	Axis4_Home_Function:MC_Home(Execute: Axis4_Home, Position: 0, HomingMode: , BufferMode: , Options: , bCalibrationCam: X0_5, Axis: Axis4)
NETWORK 5
	Axis5_Home_Function:MC_Home(Execute: Axis5_Home, Position: 0, HomingMode: , BufferMode: , Options: , bCalibrationCam: X0_8, Axis: Axis5)
NETWORK 6
	Axis6_Home_Function:MC_Home(Execute: Axis6_Home, Position: 0, HomingMode: , BufferMode: , Options: , bCalibrationCam: X0_11, Axis: Axis6)
NETWORK 7
	Axis7_Home_Function:MC_Home(Execute: Axis7_Home, Position: 0, HomingMode: , BufferMode: , Options: , bCalibrationCam: X0_14, Axis: Axis7)
NETWORK 8
	Axis8_Home_Function:MC_Home(Execute: Axis8_Home, Position: 0, HomingMode: , BufferMode: , Options: , bCalibrationCam: X1_4, Axis: Axis8)
NETWORK 9
	Axis9_Home_Function:MC_Home(Execute: Axis9_Home, Position: 0, HomingMode: , BufferMode: , Options: , bCalibrationCam: X1_7, Axis: Axis9)
NETWORK 10
	Axis10_Home_Function:MC_Home(Execute: Axis10_Home, Position: 0, HomingMode: , BufferMode: , Options: , bCalibrationCam: X1_13, Axis: Axis10)
NETWORK 11
	Axis11_Home_Function:MC_Home(Execute: Axis11_Home, Position: 0, HomingMode: , BufferMode: , Options: , bCalibrationCam: X4_9, Axis: Axis11)
NETWORK 12
	Axis12_Home_Function:MC_Home(Execute: Axis12_Home, Position: 0, HomingMode: , BufferMode: , Options: , bCalibrationCam: X4_9, Axis: Axis12)
_END_FBD_
END_PROGRAM

(* POU Other_Folder/Motion/Power_Pro, FBD *)
PROGRAM Power_Pro
VAR

END_VAR
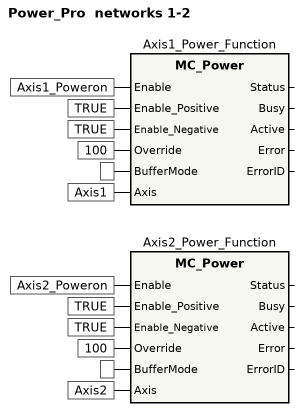
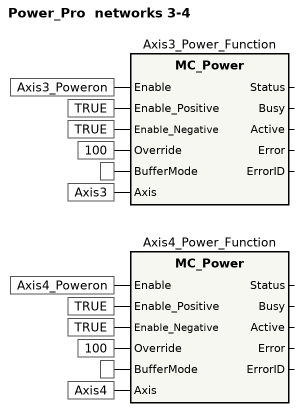
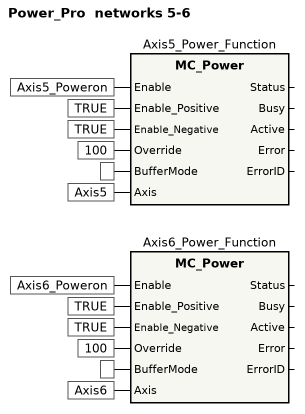
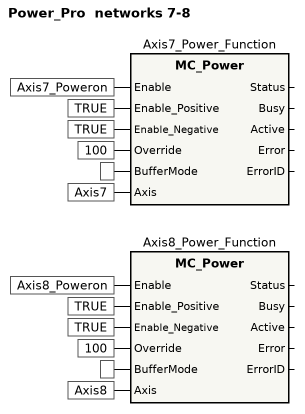
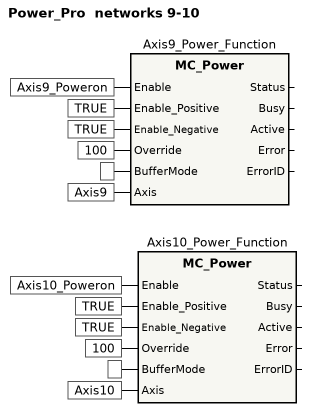
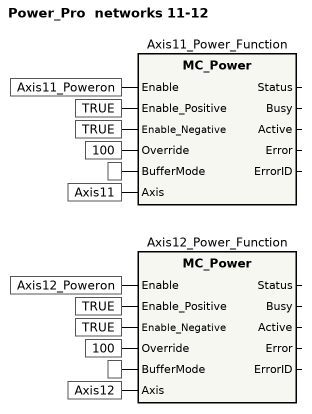
_FBD_ (* Function Block Diagram *)
NETWORK 1
	Axis1_Power_Function:MC_Power(Enable: Axis1_Poweron, Enable_Positive: TRUE, Enable_Negative: TRUE, Override: 100, BufferMode: , Axis: Axis1)
NETWORK 2
	Axis2_Power_Function:MC_Power(Enable: Axis2_Poweron, Enable_Positive: TRUE, Enable_Negative: TRUE, Override: 100, BufferMode: , Axis: Axis2)
NETWORK 3
	Axis3_Power_Function:MC_Power(Enable: Axis3_Poweron, Enable_Positive: TRUE, Enable_Negative: TRUE, Override: 100, BufferMode: , Axis: Axis3)
NETWORK 4
	Axis4_Power_Function:MC_Power(Enable: Axis4_Poweron, Enable_Positive: TRUE, Enable_Negative: TRUE, Override: 100, BufferMode: , Axis: Axis4)
NETWORK 5
	Axis5_Power_Function:MC_Power(Enable: Axis5_Poweron, Enable_Positive: TRUE, Enable_Negative: TRUE, Override: 100, BufferMode: , Axis: Axis5)
NETWORK 6
	Axis6_Power_Function:MC_Power(Enable: Axis6_Poweron, Enable_Positive: TRUE, Enable_Negative: TRUE, Override: 100, BufferMode: , Axis: Axis6)
NETWORK 7
	Axis7_Power_Function:MC_Power(Enable: Axis7_Poweron, Enable_Positive: TRUE, Enable_Negative: TRUE, Override: 100, BufferMode: , Axis: Axis7)
NETWORK 8
	Axis8_Power_Function:MC_Power(Enable: Axis8_Poweron, Enable_Positive: TRUE, Enable_Negative: TRUE, Override: 100, BufferMode: , Axis: Axis8)
NETWORK 9
	Axis9_Power_Function:MC_Power(Enable: Axis9_Poweron, Enable_Positive: TRUE, Enable_Negative: TRUE, Override: 100, BufferMode: , Axis: Axis9)
NETWORK 10
	Axis10_Power_Function:MC_Power(Enable: Axis10_Poweron, Enable_Positive: TRUE, Enable_Negative: TRUE, Override: 100, BufferMode: , Axis: Axis10)
NETWORK 11
	Axis11_Power_Function:MC_Power(Enable: Axis11_Poweron, Enable_Positive: TRUE, Enable_Negative: TRUE, Override: 100, BufferMode: , Axis: Axis11)
NETWORK 12
	Axis12_Power_Function:MC_Power(Enable: Axis12_Poweron, Enable_Positive: TRUE, Enable_Negative: TRUE, Override: 100, BufferMode: , Axis: Axis12)
_END_FBD_
END_PROGRAM

(* POU Other_Folder/Motion/Abs_Pro, FBD *)
PROGRAM Abs_Pro
VAR




END_VAR
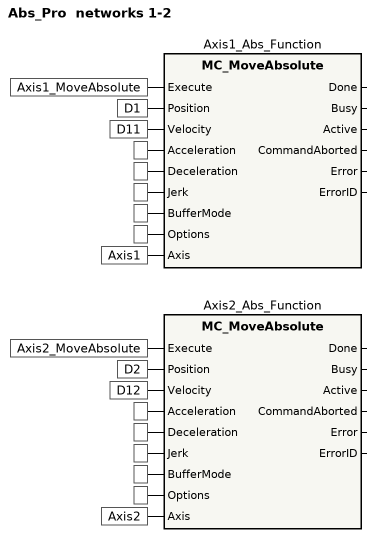
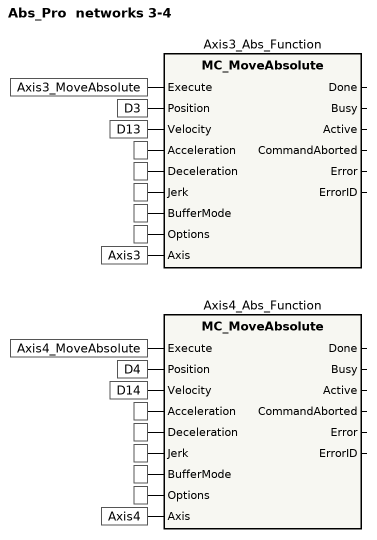
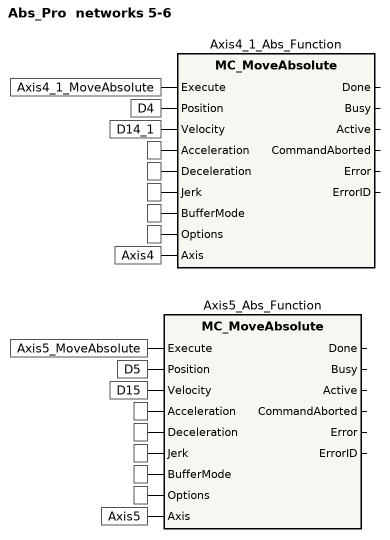
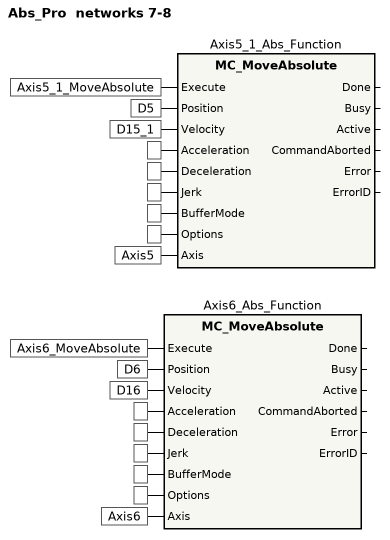
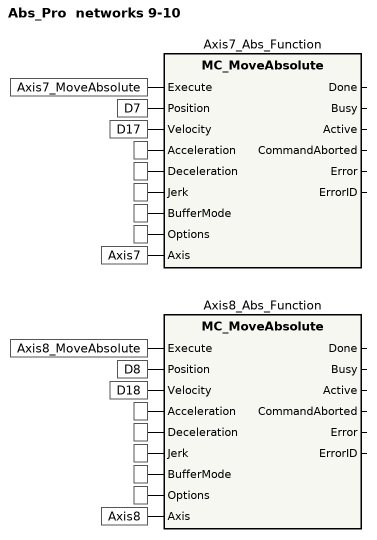
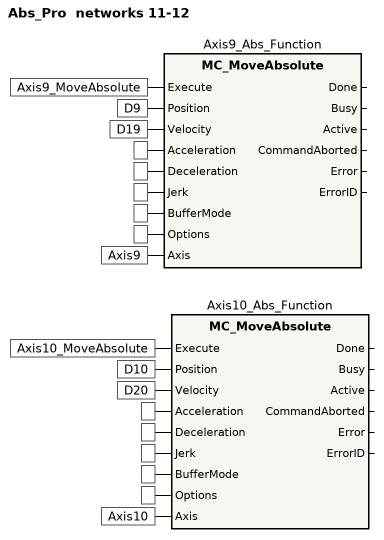
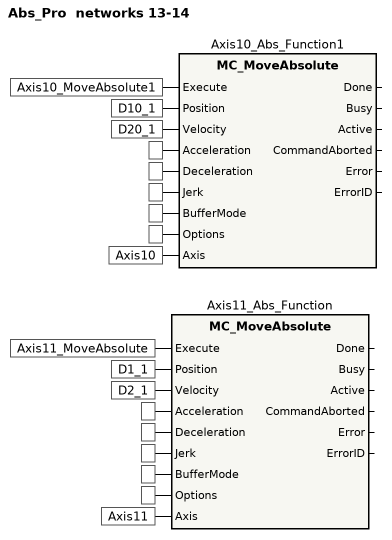
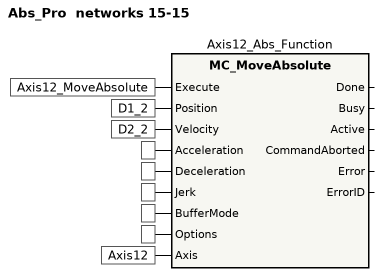
_FBD_ (* Function Block Diagram *)
NETWORK 1
	Axis1_Abs_Function:MC_MoveAbsolute(Execute: Axis1_MoveAbsolute, Position: D1, Velocity: D11, Acceleration: , Deceleration: , Jerk: , BufferMode: , Options: , Axis: Axis1)
NETWORK 2
	Axis2_Abs_Function:MC_MoveAbsolute(Execute: Axis2_MoveAbsolute, Position: D2, Velocity: D12, Acceleration: , Deceleration: , Jerk: , BufferMode: , Options: , Axis: Axis2)
NETWORK 3
	Axis3_Abs_Function:MC_MoveAbsolute(Execute: Axis3_MoveAbsolute, Position: D3, Velocity: D13, Acceleration: , Deceleration: , Jerk: , BufferMode: , Options: , Axis: Axis3)
NETWORK 4
	Axis4_Abs_Function:MC_MoveAbsolute(Execute: Axis4_MoveAbsolute, Position: D4, Velocity: D14, Acceleration: , Deceleration: , Jerk: , BufferMode: , Options: , Axis: Axis4)
NETWORK 5
	Axis4_1_Abs_Function:MC_MoveAbsolute(Execute: Axis4_1_MoveAbsolute, Position: D4, Velocity: D14_1, Acceleration: , Deceleration: , Jerk: , BufferMode: , Options: , Axis: Axis4)
NETWORK 6
	Axis5_Abs_Function:MC_MoveAbsolute(Execute: Axis5_MoveAbsolute, Position: D5, Velocity: D15, Acceleration: , Deceleration: , Jerk: , BufferMode: , Options: , Axis: Axis5)
NETWORK 7
	Axis5_1_Abs_Function:MC_MoveAbsolute(Execute: Axis5_1_MoveAbsolute, Position: D5, Velocity: D15_1, Acceleration: , Deceleration: , Jerk: , BufferMode: , Options: , Axis: Axis5)
NETWORK 8
	Axis6_Abs_Function:MC_MoveAbsolute(Execute: Axis6_MoveAbsolute, Position: D6, Velocity: D16, Acceleration: , Deceleration: , Jerk: , BufferMode: , Options: , Axis: Axis6)
NETWORK 9
	Axis7_Abs_Function:MC_MoveAbsolute(Execute: Axis7_MoveAbsolute, Position: D7, Velocity: D17, Acceleration: , Deceleration: , Jerk: , BufferMode: , Options: , Axis: Axis7)
NETWORK 10
	Axis8_Abs_Function:MC_MoveAbsolute(Execute: Axis8_MoveAbsolute, Position: D8, Velocity: D18, Acceleration: , Deceleration: , Jerk: , BufferMode: , Options: , Axis: Axis8)
NETWORK 11
	Axis9_Abs_Function:MC_MoveAbsolute(Execute: Axis9_MoveAbsolute, Position: D9, Velocity: D19, Acceleration: , Deceleration: , Jerk: , BufferMode: , Options: , Axis: Axis9)
NETWORK 12
	Axis10_Abs_Function:MC_MoveAbsolute(Execute: Axis10_MoveAbsolute, Position: D10, Velocity: D20, Acceleration: , Deceleration: , Jerk: , BufferMode: , Options: , Axis: Axis10)
NETWORK 13
	Axis10_Abs_Function1:MC_MoveAbsolute(Execute: Axis10_MoveAbsolute1, Position: D10_1, Velocity: D20_1, Acceleration: , Deceleration: , Jerk: , BufferMode: , Options: , Axis: Axis10)
NETWORK 14
	Axis11_Abs_Function:MC_MoveAbsolute(Execute: Axis11_MoveAbsolute, Position: D1_1, Velocity: D2_1, Acceleration: , Deceleration: , Jerk: , BufferMode: , Options: , Axis: Axis11)
NETWORK 15
	Axis12_Abs_Function:MC_MoveAbsolute(Execute: Axis12_MoveAbsolute, Position: D1_2, Velocity: D2_2, Acceleration: , Deceleration: , Jerk: , BufferMode: , Options: , Axis: Axis12)
_END_FBD_
END_PROGRAM

(* POU Other_Folder/Motion/Halt_Pro, FBD *)
PROGRAM Halt_Pro
VAR

END_VAR
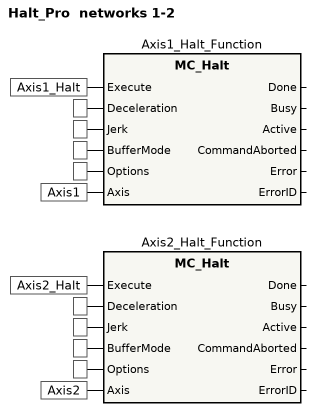
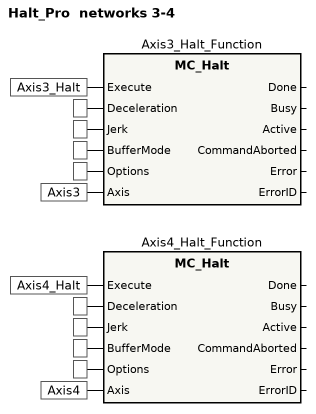
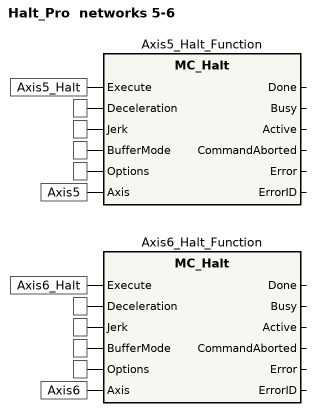
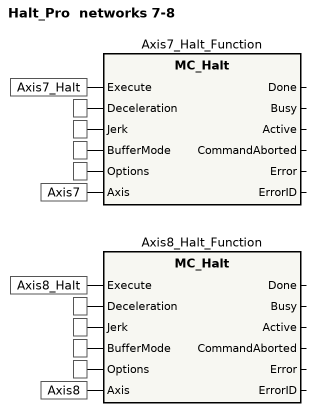
